// TwinCAT 3 PLC project PLC1
// ProgramVersion: 3.1.4024.0
// libraries:
//   CmpBitmapPool, * (System)
//   Tc2_Standard, * (Beckhoff Automation GmbH)
//   Tc2_System, * (Beckhoff Automation GmbH)
//   Tc3_Module, * (Beckhoff Automation GmbH)
// project tree:
//   GVLs/ GVL_UNIT_Blikkenvullijn.TcGVL
//   LIB/1. Control Modules/Brisq/1. DEV_Base/ FB_DeviceBase.TcPOU, stDevBase.TcDUT
//   LIB/1. Control Modules/Brisq/2. DEV_AnaIn/ FB_DEV_AnaIn.TcPOU, ITF_DEV_AnaIn.TcIO
//   LIB/1. Control Modules/Brisq/3. DEV_DigIn/ FB_DEV_DigIn.TcPOU, ITF_DigIn.TcIO
//   LIB/1. Control Modules/Brisq/4. DEV_Valve/ DEV_Valve.TcPOU, ITF_Valve.TcIO
//   LIB/1. Control Modules/Brisq/4. DEV_Valve/ENUMs/ E_ValveState.TcDUT
//   LIB/1. Control Modules/Brisq/4. DEV_Valve/STRUCTs/ stDevValve.TcDUT
//   LIB/1. Control Modules/Brisq/5. DEV_ControlValve/ DEV_CtrlValve.TcPOU, ITF_ControlValve.TcIO
//   LIB/1. Control Modules/Brisq/5. DEV_ControlValve/ENUMs/ E_CtrlValveState.TcDUT
//   LIB/1. Control Modules/Brisq/6. DEV_Motor/ENUMs/ E_MotorState.TcDUT
//   LIB/1. Control Modules/Brisq/6. DEV_Motor/ ITF_Motor_1.TcIO
//   LIB/1. Control Modules/Brisq/ENUMs/ E_OperationMode.TcDUT
//   LIB/1. Control Modules/Brisq/ FB_Devices.TcPOU
//   LIB/2. Equipment Modules/1. FB_Base/ FB_EMbase.TcPOU, stEMbase.TcDUT
//   LIB/2. Equipment Modules/2. EM_Machine_PackML/ FB_Machine_PackML.TcPOU, ITF_PackML.TcIO, STRUCT_Machine_PackML.TcDUT
//   LIB/3. Units/1. UN_Base/ FB_UN_base.TcPOU, stUNbase.TcDUT
//   / PlcTask.TcTTO
//   POUs/1. Control Modules/1. CM_Motor/ CM_Motor.TcPOU, ITF_Motor.TcIO
//   POUs/1. Control Modules/1. CM_Motor/Enums/ E_Motor_Error_State.TcDUT, E_Motor_State.TcDUT
//   POUs/1. Control Modules/1. CM_Motor/Structs/1. CS/ CM_Motor_CS.TcDUT
//   POUs/1. Control Modules/1. CM_Motor/Structs/2. HMI/ CM_Motor_HMI.TcDUT
//   POUs/1. Control Modules/1. CM_Motor/Structs/3. STS/ CM_Motor_STS.TcDUT
//   POUs/1. Control Modules/1. CM_Motor/Structs/4. ALM/ CM_Motor_ALM.TcDUT
//   POUs/1. Control Modules/1. CM_Motor/Structs/5. WRN/ CM_Motor_WRN.TcDUT
//   POUs/1. Control Modules/1. CM_Motor/Structs/6. PAR/ CM_Motor_PAR.TcDUT
//   POUs/1. Control Modules/1. CM_Motor/Structs/7. SIM/ CM_Motor_SIM.TcDUT
//   POUs/1. Control Modules/1. CM_Motor/Structs/ STRUCT_CM_Motor.TcDUT
//   POUs/1. Control Modules/2. CM_Sensor/ CM_Sensor.TcPOU, ITF_Sensor.TcIO
//   POUs/1. Control Modules/2. CM_Sensor/Structs/1. CS/ CM_Sensor_CS.TcDUT
//   POUs/1. Control Modules/2. CM_Sensor/Structs/2. HMI/ CM_Sensor_HMI.TcDUT
//   POUs/1. Control Modules/2. CM_Sensor/Structs/3. STS/ CM_Sensor_STS.TcDUT
//   POUs/1. Control Modules/2. CM_Sensor/Structs/4. ALM/ CM_Sensor_ALM.TcDUT
//   POUs/1. Control Modules/2. CM_Sensor/Structs/5. WRN/ CM_Sensor_WRN.TcDUT
//   POUs/1. Control Modules/2. CM_Sensor/Structs/6. PAR/ CM_Sensor_PAR.TcDUT
//   POUs/1. Control Modules/2. CM_Sensor/Structs/7. SIM/ CM_Sensor_SIM.TcDUT
//   POUs/1. Control Modules/2. CM_Sensor/Structs/ STRUCT_CM_Sensor.TcDUT
//   POUs/1. Control Modules/4. CM_Valve/ CM_Valve.TcPOU, ITF_Valve2.TcIO
//   POUs/1. Control Modules/4. CM_Valve/Enums/ E_Valve_Error_State.TcDUT, E_Valve_State.TcDUT
//   POUs/1. Control Modules/4. CM_Valve/Structs/1. CS/ CM_Valve_CS.TcDUT
//   POUs/1. Control Modules/4. CM_Valve/Structs/2. HMI/ CM_Valve_HMI.TcDUT
//   POUs/1. Control Modules/4. CM_Valve/Structs/3. STS/ CM_Valve_STS.TcDUT
//   POUs/1. Control Modules/4. CM_Valve/Structs/4. ALM/ CM_Valve_ALM.TcDUT
//   POUs/1. Control Modules/4. CM_Valve/Structs/5. WRN/ CM_Valve_WRN.TcDUT
//   POUs/1. Control Modules/4. CM_Valve/Structs/6. PAR/ CM_Valve_PAR.TcDUT
//   POUs/1. Control Modules/4. CM_Valve/Structs/7. SIM/ CM_Valve_SIM.TcDUT
//   POUs/1. Control Modules/4. CM_Valve/Structs/ STRUCT_CM_Valve.TcDUT
//   POUs/2. Equipment Modules/1. EM_Can_Supply/Enums/ E_State_Can_Supply.TcDUT
//   POUs/2. Equipment Modules/1. EM_Can_Supply/ EM_Can_Supply.TcPOU, ITF_Can_Supply.TcIO
//   POUs/2. Equipment Modules/1. EM_Can_Supply/Structs/1. CS/ EM_CanSupply_CS.TcDUT
//   POUs/2. Equipment Modules/1. EM_Can_Supply/Structs/2. HMI/ EM_CanSupply_HMI.TcDUT
//   POUs/2. Equipment Modules/1. EM_Can_Supply/Structs/3. STS/ EM_CanSupply_STS.TcDUT
//   POUs/2. Equipment Modules/1. EM_Can_Supply/Structs/4. ALM/ EM_CanSupply_ALM.TcDUT
//   POUs/2. Equipment Modules/1. EM_Can_Supply/Structs/5. WRN/ EM_CanSupply_WRN.TcDUT
//   POUs/2. Equipment Modules/1. EM_Can_Supply/Structs/6. PAR/ EM_CanSupply_PAR.TcDUT
//   POUs/2. Equipment Modules/1. EM_Can_Supply/Structs/7. SIM/ EM_CanSupply_SIM.TcDUT
//   POUs/2. Equipment Modules/1. EM_Can_Supply/Structs/ STRUCT_EM_CanSupply.TcDUT
//   POUs/2. Equipment Modules/2. EM_Filling/ EM_Filling.TcPOU
//   POUs/2. Equipment Modules/2. EM_Filling/Enums/ E_State_Filling.TcDUT
//   POUs/2. Equipment Modules/2. EM_Filling/Structs/1. CS/ EM_Filling_CS.TcDUT
//   POUs/2. Equipment Modules/2. EM_Filling/Structs/2. HMI/ EM_Filling_HMI.TcDUT
//   POUs/2. Equipment Modules/2. EM_Filling/Structs/3. STS/ EM_Filling_STS.TcDUT
//   POUs/2. Equipment Modules/2. EM_Filling/Structs/4. ALM/ EM_Filling_ALM.TcDUT
//   POUs/2. Equipment Modules/2. EM_Filling/Structs/5. WRN/ EM_Filling_WRN.TcDUT
//   POUs/2. Equipment Modules/2. EM_Filling/Structs/6. PAR/ EM_Filling_PAR.TcDUT
//   POUs/2. Equipment Modules/2. EM_Filling/Structs/7. SIM/ EM_Filling_SIM.TcDUT
//   POUs/2. Equipment Modules/2. EM_Filling/Structs/ STRUCT_EM_Filling.TcDUT
//   POUs/2. Equipment Modules/4. EM_Transport/ EM_Transport.TcPOU, ITF_EM_Transport.TcIO
//   POUs/2. Equipment Modules/4. EM_Transport/Structs/1. CS/ EM_Transport_CS.TcDUT
//   POUs/2. Equipment Modules/4. EM_Transport/Structs/2. HMI/ EM_Transport_HMI.TcDUT
//   POUs/2. Equipment Modules/4. EM_Transport/Structs/3. STS/ EM_Transport_STS.TcDUT
//   POUs/2. Equipment Modules/4. EM_Transport/Structs/4. ALM/ EM_Transport_ALM.TcDUT
//   POUs/2. Equipment Modules/4. EM_Transport/Structs/5. WRN/ EM_Transport_WRN.TcDUT
//   POUs/2. Equipment Modules/4. EM_Transport/Structs/6. PAR/ EM_Transport_PAR.TcDUT
//   POUs/2. Equipment Modules/4. EM_Transport/Structs/7. SIM/ EM_Transport_SIM.TcDUT
//   POUs/2. Equipment Modules/4. EM_Transport/Structs/ STRUCT_EM_Transport.TcDUT
//   POUs/2. Equipment Modules/3. EM_Machine/ EM_Machine.TcPOU
//   POUs/2. Equipment Modules/3. EM_Machine/Structs/1. CS/ EM_Machine_CS.TcDUT
//   POUs/2. Equipment Modules/3. EM_Machine/Structs/2. HMI/ EM_Machine_HMI.TcDUT
//   POUs/2. Equipment Modules/3. EM_Machine/Structs/3. STS/ EM_Machine_STS.TcDUT
//   POUs/2. Equipment Modules/3. EM_Machine/Structs/4. ALM/ EM_Machine_ALM.TcDUT
//   POUs/2. Equipment Modules/3. EM_Machine/Structs/5. WRN/ EM_Machine_WRN.TcDUT
//   POUs/2. Equipment Modules/3. EM_Machine/Structs/6. PAR/ EM_Machine_PAR.TcDUT
//   POUs/2. Equipment Modules/3. EM_Machine/Structs/7. SIM/ EM_Machine_SIM.TcDUT
//   POUs/2. Equipment Modules/3. EM_Machine/Structs/ STRUCT_EM_Machine.TcDUT
//   POUs/2. Equipment Modules/5. EM_Transport_Mechanische_Stop/ EM_Transport_Mechanische_Stop.TcPOU, ITF_EM_Transport_Mechanische_Stop.TcIO
//   POUs/2. Equipment Modules/5. EM_Transport_Mechanische_Stop/Enums/ E_Mechanische_Stop.TcDUT
//   POUs/2. Equipment Modules/5. EM_Transport_Mechanische_Stop/Structs/1. CS/ EM_Transport_Mechanische_Stop_CS.TcDUT
//   POUs/2. Equipment Modules/5. EM_Transport_Mechanische_Stop/Structs/2. HMI/ EM_Transport_Mechanische_Stop_HMI.TcDUT
//   POUs/2. Equipment Modules/5. EM_Transport_Mechanische_Stop/Structs/3. STS/ EM_Transport_Mechanische_Stop_STS.TcDUT
//   POUs/2. Equipment Modules/5. EM_Transport_Mechanische_Stop/Structs/4. ALM/ EM_Transport_Mechanische_Stop_ALM.TcDUT
//   POUs/2. Equipment Modules/5. EM_Transport_Mechanische_Stop/Structs/5. WRN/ EM_Transport_Mechanische_Stop_WRN.TcDUT
//   POUs/2. Equipment Modules/5. EM_Transport_Mechanische_Stop/Structs/6. PAR/ EM_Transport_Mechanische_Stop_PAR.TcDUT
//   POUs/2. Equipment Modules/5. EM_Transport_Mechanische_Stop/Structs/7. SIM/ EM_Transport_Mechanische_Stop_SIM.TcDUT
//   POUs/2. Equipment Modules/5. EM_Transport_Mechanische_Stop/Structs/ STRUCT_EM_Mechanische_Stop.TcDUT
//   POUs/3. Units/1. Unit_Blikkenvullijn/ ITF_UNIT_Blikkenvullijn.TcIO, UNIT_Blikkenvullijn.TcPOU
//   POUs/3. Units/1. Unit_Blikkenvullijn/Structs/4. ALM/ UNIT_Blikkenvullijn_ALM.TcDUT
//   POUs/3. Units/1. Unit_Blikkenvullijn/Structs/1. CS/ UNIT_Blikkenvullijn_CS.TcDUT
//   POUs/3. Units/1. Unit_Blikkenvullijn/Structs/2. HMI/ UNIT_Blikkenvullijn_HMI.TcDUT
//   POUs/3. Units/1. Unit_Blikkenvullijn/Structs/6. PAR/ UNIT_Blikkenvullijn_PAR.TcDUT
//   POUs/3. Units/1. Unit_Blikkenvullijn/Structs/7. SIM/ UNIT_Blikkenvullijn_SIM.TcDUT
//   POUs/3. Units/1. Unit_Blikkenvullijn/Structs/ STRUCT_UNIT_Blikkenvullijn.TcDUT
//   POUs/3. Units/1. Unit_Blikkenvullijn/Structs/3. STS/ UNIT_Blikkenvullijn_STS.TcDUT
//   POUs/3. Units/1. Unit_Blikkenvullijn/Structs/5. WRN/ UNIT_Blikkenvullijn_WRN.TcDUT
//   POUs/4. Management/1. AlarmHandler/ AlarmHandler.TcPOU, stErrorHandling.TcDUT
//   POUs/4. Management/2. ModeSelect/ ITF_ModeSelect.TcIO, ModeSelect.TcPOU, STRUCT_ModeSelect.TcDUT
//   POUs/4. Management/3. PackML/ E_State_PackML.TcDUT, ITF_PackMLV2.TcIO, PackML_StateMachine.TcPOU
//   POUs/ MAIN.TcPOU
// real-time tasks:
//   TASK PlcTask: cycle T#10ms, priority 20, ADS port 350

CONFIGURATION PLC1
    RESOURCE PLC ON TwinCAT3
        TASK PlcTask(INTERVAL := T#1ms, PRIORITY := 11);
        PROGRAM MAIN WITH PlcTask : MAIN;
    END_RESOURCE
END_CONFIGURATION

// ---- LIB/1. Control Modules/Brisq/1. DEV_Base/stDevBase.TcDUT
TYPE stDevBase :
STRUCT
	sTagName : STRING;
	sDescription : STRING;
END_STRUCT
END_TYPE

// ---- LIB/1. Control Modules/Brisq/4. DEV_Valve/ENUMs/E_ValveState.TcDUT
{attribute 'qualified_only'}
{attribute 'strict'}
TYPE E_ValveState :
(
	Unknown := 0,
	Open := 1,
	Closed := 2,
	Opening := 3,
	Closing := 4,
	Error := -1
);
END_TYPE

// ---- LIB/1. Control Modules/Brisq/4. DEV_Valve/STRUCTs/stDevValve.TcDUT
TYPE stDevValve :
STRUCT
	//Input to HMI
	bGetHmiError : BOOL;  //True = error
	bGetHmiStatus : BOOL; //True = Open || False = Closed
	eGetState : E_ValveState;
	eGetMode : E_OperationMode;
	
	//Output from HMI
	eSetMode : E_OperationMode; 
END_STRUCT
END_TYPE

// ---- LIB/1. Control Modules/Brisq/5. DEV_ControlValve/ENUMs/E_CtrlValveState.TcDUT
{attribute 'qualified_only'}
{attribute 'strict'}
TYPE E_CtrlValveState :
(
	Unknown := 0,
	InPosition := 1,
	Moving := 2,
	Error := -1
);
END_TYPE

// ---- LIB/1. Control Modules/Brisq/6. DEV_Motor/ENUMs/E_MotorState.TcDUT
{attribute 'qualified_only'}
{attribute 'strict'}
TYPE E_MotorState :
(
	Unknown := 0,
	Running := 1,
	Stalled := 2,
	SpeedingUp := 3,
	SpeedingDown := 4,
	Error := -1
);
END_TYPE

// ---- LIB/1. Control Modules/Brisq/ENUMs/E_OperationMode.TcDUT
{attribute 'qualified_only'}
{attribute 'strict'}
TYPE E_OperationMode :
(
	Off := 0,
	Manual := 1,
	Automatic := 2
);
END_TYPE

// ---- LIB/2. Equipment Modules/1. FB_Base/stEMbase.TcDUT
TYPE stEMbase :
STRUCT
	sTagName : STRING;
	sDescription : STRING;
END_STRUCT
END_TYPE

// ---- LIB/2. Equipment Modules/2. EM_Machine_PackML/STRUCT_Machine_PackML.TcDUT
TYPE STRUCT_Machine_PackML :
STRUCT
	//Properties
	State 			: E_State_PackML;
	//Methods
   	Abort 			: BOOL;
	Aborting_SC 	: BOOL;
	Clear 			: BOOL;
	Clearing_SC 	: BOOL;
	Execute_SC 		: BOOL;
	Completing_SC	: BOOL;
	Hold 			: BOOL;
	Holding_SC 		: BOOL;
	Reset 			: BOOL;
	Resetting_SC 	: BOOL;
	Start 			: BOOL;
	Starting_SC 	: BOOL;
	Stop 			: BOOL;
	Stopping_SC 	: BOOL;
	Suspend 		: BOOL;
	Suspending_SC 	: BOOL;
	Unhold 			: BOOL;
	Unholding_SC 	: BOOL;
	Unsuspend 		: BOOL;
	Unsuspending_SC : BOOL;
END_STRUCT
END_TYPE

// ---- LIB/3. Units/1. UN_Base/stUNbase.TcDUT
TYPE stUNbase :
STRUCT
	sTagName : STRING;
	sDescription : STRING;
END_STRUCT
END_TYPE

// ---- POUs/1. Control Modules/1. CM_Motor/Enums/E_Motor_Error_State.TcDUT
{attribute 'qualified_only'}
{attribute 'strict'}
TYPE E_Motor_Error_State :
(
	enum_member := 0
);
END_TYPE

// ---- POUs/1. Control Modules/1. CM_Motor/Enums/E_Motor_State.TcDUT
{attribute 'qualified_only'}
{attribute 'strict'}
TYPE E_Motor_State :
(
	enum_member := 0
);
END_TYPE

// ---- POUs/1. Control Modules/1. CM_Motor/Structs/1. CS/CM_Motor_CS.TcDUT
TYPE CM_Motor_CS :
STRUCT
	Start		: BOOL;
	Stop		: BOOL;
	Reset		: BOOL;
	Abort		: BOOL;
	Clear		: BOOL;
	UnSuspend	: BOOL;
	Suspend		: BOOL;
	UnHold		: BOOL;
	Hold		: BOOL;
	Richting_L	: BOOL;
	Richting_R	: BOOL;
	Toerental	: INT;
	Auto		: BOOL;
	Manueel		: BOOL;
END_STRUCT
END_TYPE

// ---- POUs/1. Control Modules/1. CM_Motor/Structs/2. HMI/CM_Motor_HMI.TcDUT
TYPE CM_Motor_HMI :
STRUCT
	Start		: BOOL;
	Stop		: BOOL;
	Reset		: BOOL;
	Abort		: BOOL;
	Clear		: BOOL;
	UnSuspend	: BOOL;
	Suspend		: BOOL;
	UnHold		: BOOL;
	Hold		: BOOL;
	Richting_L	: BOOL;
	Richting_R	: BOOL;
	Toerental	: INT;
	Auto		: BOOL;
	Manueel		: BOOL;
END_STRUCT
END_TYPE

// ---- POUs/1. Control Modules/1. CM_Motor/Structs/3. STS/CM_Motor_STS.TcDUT
TYPE CM_Motor_STS :
STRUCT
	Tag				: STRING;
	State 			: E_State_PackML;
	Error_State 	: E_Motor_Error_State;
	Richting_L		: BOOL;
	Richting_R		: BOOL;
	Auto			: BOOL;
	Manueel			: BOOL;
	Toerental 		: INT;
	
	Starting_SC		: BOOL;
	Execute_SC		: BOOL;
	Resetting_SC	: BOOL;
	Holding_SC		: BOOL;
	Unholding_SC	: BOOL;
	Suspending_SC	: BOOL;
	Unsuspending_SC	: BOOL;
	Aborting_SC		: BOOL;
	Clearing_SC		: BOOL;
	Stopping_SC		: BOOL;
	Completing_SC	: BOOL;
END_STRUCT
END_TYPE

// ---- POUs/1. Control Modules/1. CM_Motor/Structs/4. ALM/CM_Motor_ALM.TcDUT
TYPE CM_Motor_ALM :
STRUCT
END_STRUCT
END_TYPE

// ---- POUs/1. Control Modules/1. CM_Motor/Structs/5. WRN/CM_Motor_WRN.TcDUT
TYPE CM_Motor_WRN :
STRUCT
END_STRUCT
END_TYPE

// ---- POUs/1. Control Modules/1. CM_Motor/Structs/6. PAR/CM_Motor_PAR.TcDUT
TYPE CM_Motor_PAR :
STRUCT
END_STRUCT
END_TYPE

// ---- POUs/1. Control Modules/1. CM_Motor/Structs/7. SIM/CM_Motor_SIM.TcDUT
TYPE CM_Motor_SIM :
STRUCT
END_STRUCT
END_TYPE

// ---- POUs/1. Control Modules/1. CM_Motor/Structs/STRUCT_CM_Motor.TcDUT
TYPE STRUCT_CM_Motor :
STRUCT
	CS	: CM_Motor_CS;
	HMI	: CM_Motor_HMI;
	STS	: CM_Motor_STS;
	ALM	: CM_Motor_ALM;
	WRN	: CM_Motor_WRN;
	PAR	: CM_Motor_PAR;
	SIM	: CM_Motor_SIM;
END_STRUCT
END_TYPE

// ---- POUs/1. Control Modules/2. CM_Sensor/Structs/1. CS/CM_Sensor_CS.TcDUT
TYPE CM_Sensor_CS :
STRUCT
	Auto		: BOOL;
	Manueel		: BOOL;
	Output		: BOOL;
END_STRUCT
END_TYPE

// ---- POUs/1. Control Modules/2. CM_Sensor/Structs/2. HMI/CM_Sensor_HMI.TcDUT
TYPE CM_Sensor_HMI :
STRUCT
	Auto		: BOOL;
	Manueel		: BOOL;
	Output		: BOOL;
END_STRUCT
END_TYPE

// ---- POUs/1. Control Modules/2. CM_Sensor/Structs/3. STS/CM_Sensor_STS.TcDUT
TYPE CM_Sensor_STS :
STRUCT
	Tag				: STRING;
	Output			: BOOL;
	Auto			: BOOL;
	Manueel			: BOOL;
END_STRUCT
END_TYPE

// ---- POUs/1. Control Modules/2. CM_Sensor/Structs/4. ALM/CM_Sensor_ALM.TcDUT
TYPE CM_Sensor_ALM :
STRUCT
END_STRUCT
END_TYPE

// ---- POUs/1. Control Modules/2. CM_Sensor/Structs/5. WRN/CM_Sensor_WRN.TcDUT
TYPE CM_Sensor_WRN :
STRUCT
END_STRUCT
END_TYPE

// ---- POUs/1. Control Modules/2. CM_Sensor/Structs/6. PAR/CM_Sensor_PAR.TcDUT
TYPE CM_Sensor_PAR :
STRUCT
END_STRUCT
END_TYPE

// ---- POUs/1. Control Modules/2. CM_Sensor/Structs/7. SIM/CM_Sensor_SIM.TcDUT
TYPE CM_Sensor_SIM :
STRUCT
END_STRUCT
END_TYPE

// ---- POUs/1. Control Modules/2. CM_Sensor/Structs/STRUCT_CM_Sensor.TcDUT
TYPE STRUCT_CM_Sensor :
STRUCT
	CS	: CM_Sensor_CS;
	HMI	: CM_Sensor_HMI;
	STS	: CM_Sensor_STS;
	ALM	: CM_Sensor_ALM;
	WRN	: CM_Sensor_WRN;
	PAR	: CM_Sensor_PAR;
	SIM	: CM_Sensor_SIM;
END_STRUCT
END_TYPE

// ---- POUs/1. Control Modules/4. CM_Valve/Enums/E_Valve_Error_State.TcDUT
{attribute 'qualified_only'}
{attribute 'strict'}
TYPE E_Valve_Error_State :
(
	enum_member := 0
);
END_TYPE

// ---- POUs/1. Control Modules/4. CM_Valve/Enums/E_Valve_State.TcDUT
{attribute 'qualified_only'}
{attribute 'strict'}
TYPE E_Valve_State :
(
	enum_member := 0
);
END_TYPE

// ---- POUs/1. Control Modules/4. CM_Valve/Structs/1. CS/CM_Valve_CS.TcDUT
TYPE CM_Valve_CS :
STRUCT
	Start		: BOOL;
	Stop		: BOOL;
	Reset		: BOOL;
	Abort		: BOOL;
	Clear		: BOOL;
	UnSuspend	: BOOL;
	Suspend		: BOOL;
	UnHold		: BOOL;
	Hold		: BOOL;
	Auto		: BOOL;
	Manueel		: BOOL;
	Open		: BOOL;
	Close		: BOOL;
END_STRUCT
END_TYPE

// ---- POUs/1. Control Modules/4. CM_Valve/Structs/2. HMI/CM_Valve_HMI.TcDUT
TYPE CM_Valve_HMI :
STRUCT
	Start		: BOOL;
	Stop		: BOOL;
	Reset		: BOOL;
	Abort		: BOOL;
	Clear		: BOOL;
	UnSuspend	: BOOL;
	Suspend		: BOOL;
	UnHold		: BOOL;
	Hold		: BOOL;
	Auto		: BOOL;
	Manueel		: BOOL;
	Open		: BOOL;
	Close		: BOOL;
END_STRUCT
END_TYPE

// ---- POUs/1. Control Modules/4. CM_Valve/Structs/3. STS/CM_Valve_STS.TcDUT
TYPE CM_Valve_STS :
STRUCT
	Tag				: STRING;
	State 			: E_State_PackML;
	Error_State 	: E_Motor_Error_State;
	Auto			: BOOL;
	Manueel			: BOOL;
	Open			: BOOL;
	Close			: BOOL;
	
	Starting_SC		: BOOL;
	Execute_SC		: BOOL;
	Resetting_SC	: BOOL;
	Holding_SC		: BOOL;
	Unholding_SC	: BOOL;
	Suspending_SC	: BOOL;
	Unsuspending_SC	: BOOL;
	Aborting_SC		: BOOL;
	Clearing_SC		: BOOL;
	Stopping_SC		: BOOL;
	Completing_SC	: BOOL;
END_STRUCT
END_TYPE

// ---- POUs/1. Control Modules/4. CM_Valve/Structs/4. ALM/CM_Valve_ALM.TcDUT
TYPE CM_Valve_ALM :
STRUCT
END_STRUCT
END_TYPE

// ---- POUs/1. Control Modules/4. CM_Valve/Structs/5. WRN/CM_Valve_WRN.TcDUT
TYPE CM_Valve_WRN :
STRUCT
END_STRUCT
END_TYPE

// ---- POUs/1. Control Modules/4. CM_Valve/Structs/6. PAR/CM_Valve_PAR.TcDUT
TYPE CM_Valve_PAR :
STRUCT
END_STRUCT
END_TYPE

// ---- POUs/1. Control Modules/4. CM_Valve/Structs/7. SIM/CM_Valve_SIM.TcDUT
TYPE CM_Valve_SIM :
STRUCT
END_STRUCT
END_TYPE

// ---- POUs/1. Control Modules/4. CM_Valve/Structs/STRUCT_CM_Valve.TcDUT
TYPE STRUCT_CM_Valve :
STRUCT
	CS	: CM_Valve_CS;
	HMI	: CM_Valve_HMI;
	STS	: CM_Valve_STS;
	ALM	: CM_Valve_ALM;
	WRN	: CM_Valve_WRN;
	PAR	: CM_Valve_PAR;
	SIM	: CM_Valve_SIM;
END_STRUCT
END_TYPE

// ---- POUs/2. Equipment Modules/1. EM_Can_Supply/Enums/E_State_Can_Supply.TcDUT
{attribute 'qualified_only'}
{attribute 'strict'}
TYPE E_State_Can_Supply :
(
	State := 0
);
END_TYPE

// ---- POUs/2. Equipment Modules/1. EM_Can_Supply/Structs/1. CS/EM_CanSupply_CS.TcDUT
TYPE EM_CanSupply_CS :
STRUCT
	Start		: BOOL;
	Stop		: BOOL;
	Reset		: BOOL;
	Abort		: BOOL;
	Richting_L	: BOOL;
	Richting_R	: BOOL;
	Toerental	: INT;
	Auto		: BOOL;
	Manueel		: BOOL;
	Clear		: BOOL;
	UnSuspend	: BOOL;
	Suspend		: BOOL;
	UnHold		: BOOL;
	Hold		: BOOL;
END_STRUCT
END_TYPE

// ---- POUs/2. Equipment Modules/1. EM_Can_Supply/Structs/2. HMI/EM_CanSupply_HMI.TcDUT
TYPE EM_CanSupply_HMI :
STRUCT
	Start		: BOOL;
	Stop		: BOOL;
	Reset		: BOOL;
	Abort		: BOOL;
	Richting_L	: BOOL;
	Richting_R	: BOOL;
	Toerental	: INT;
	Auto		: BOOL;
	Manueel		: BOOL;
END_STRUCT
END_TYPE

// ---- POUs/2. Equipment Modules/1. EM_Can_Supply/Structs/3. STS/EM_CanSupply_STS.TcDUT
TYPE EM_CanSupply_STS :
STRUCT
	Tag				: STRING;
	State 			: E_State_PackML;
	StringState		: STRING;
	Error_State 	: E_Motor_Error_State;
	Auto			: BOOL;
	Manueel			: BOOL;
	Richting_L		: BOOL;
	Richting_R		: BOOL;
	Starting_SC 	: BOOL;
	Execute_SC 		: BOOL;
	Resetting_SC 	: BOOL;
	Holding_SC 		: BOOL;
	Unholding_SC 	: BOOL;
	Suspending_SC	: BOOL;
	Unsuspending_SC	: BOOL;
	Aborting_SC		: BOOL;
	Clearing_SC		: BOOL;
	Stopping_SC		: BOOL;
	Completing_SC	: BOOL;
END_STRUCT
END_TYPE

// ---- POUs/2. Equipment Modules/1. EM_Can_Supply/Structs/4. ALM/EM_CanSupply_ALM.TcDUT
TYPE EM_CanSupply_ALM :
STRUCT
END_STRUCT
END_TYPE

// ---- POUs/2. Equipment Modules/1. EM_Can_Supply/Structs/5. WRN/EM_CanSupply_WRN.TcDUT
TYPE EM_CanSupply_WRN :
STRUCT
END_STRUCT
END_TYPE

// ---- POUs/2. Equipment Modules/1. EM_Can_Supply/Structs/6. PAR/EM_CanSupply_PAR.TcDUT
TYPE EM_CanSupply_PAR :
STRUCT
END_STRUCT
END_TYPE

// ---- POUs/2. Equipment Modules/1. EM_Can_Supply/Structs/7. SIM/EM_CanSupply_SIM.TcDUT
TYPE EM_CanSupply_SIM :
STRUCT
	Sen_A1_Near_TRUE	: BOOL;
	Sen_A1_Far_TRUE		: BOOL;
	Sen_A2_Near_TRUE	: BOOL;
	Sen_A2_Far_TRUE		: BOOL;
END_STRUCT
END_TYPE

// ---- POUs/2. Equipment Modules/1. EM_Can_Supply/Structs/STRUCT_EM_CanSupply.TcDUT
TYPE STRUCT_EM_CanSupply :
STRUCT
	CS	: EM_CanSupply_CS;
	HMI	: EM_CanSupply_HMI;
	STS	: EM_CanSupply_STS;
	ALM	: EM_CanSupply_ALM;
	WRN	: EM_CanSupply_WRN;
	PAR	: EM_CanSupply_PAR;
	SIM	: EM_CanSupply_SIM;	
END_STRUCT
END_TYPE

// ---- POUs/2. Equipment Modules/2. EM_Filling/Enums/E_State_Filling.TcDUT
{attribute 'qualified_only'}
{attribute 'strict'}
TYPE E_State_Filling :
(
	State := 0
);
END_TYPE

// ---- POUs/2. Equipment Modules/2. EM_Filling/Structs/1. CS/EM_Filling_CS.TcDUT
TYPE EM_Filling_CS :
STRUCT
	Start		: BOOL;
	Stop		: BOOL;
	Reset		: BOOL;
	Abort		: BOOL;
	Richting_L	: BOOL;
	Richting_R	: BOOL;
	Toerental	: INT;
	Auto		: BOOL;
	Manueel		: BOOL;
	Clear		: BOOL;
	UnSuspend	: BOOL;
	Suspend		: BOOL;
	UnHold		: BOOL;
	Hold		: BOOL;
END_STRUCT
END_TYPE

// ---- POUs/2. Equipment Modules/2. EM_Filling/Structs/2. HMI/EM_Filling_HMI.TcDUT
TYPE EM_Filling_HMI :
STRUCT
	Start		: BOOL;
	Stop		: BOOL;
	Reset		: BOOL;
	Abort		: BOOL;
	Richting_L	: BOOL;
	Richting_R	: BOOL;
	Toerental	: INT;
	Auto		: BOOL;
	Manueel		: BOOL;
	Clear		: BOOL;
	UnSuspend	: BOOL;
	Suspend		: BOOL;
	UnHold		: BOOL;
	Hold		: BOOL;
END_STRUCT
END_TYPE

// ---- POUs/2. Equipment Modules/2. EM_Filling/Structs/3. STS/EM_Filling_STS.TcDUT
TYPE EM_Filling_STS :
STRUCT
	Tag				: STRING;
	State 			: E_State_PackML;
	StringState		: STRING;
	Error_State 	: E_Motor_Error_State;
	Richting_L		: BOOL;
	Richting_R		: BOOL;
	Auto 			: BOOL;
	Manueel 		: BOOL;
	Starting_SC 	: BOOL;
	Execute_SC 		: BOOL;
	Resetting_SC 	: BOOL;
	Holding_SC 		: BOOL;
	Unholding_SC 	: BOOL;
	Suspending_SC	: BOOL;
	Unsuspending_SC	: BOOL;
	Aborting_SC		: BOOL;
	Clearing_SC		: BOOL;
	Stopping_SC		: BOOL;
	Completing_SC	: BOOL;
END_STRUCT
END_TYPE

// ---- POUs/2. Equipment Modules/2. EM_Filling/Structs/4. ALM/EM_Filling_ALM.TcDUT
TYPE EM_Filling_ALM :
STRUCT
END_STRUCT
END_TYPE

// ---- POUs/2. Equipment Modules/2. EM_Filling/Structs/5. WRN/EM_Filling_WRN.TcDUT
TYPE EM_Filling_WRN :
STRUCT
END_STRUCT
END_TYPE

// ---- POUs/2. Equipment Modules/2. EM_Filling/Structs/6. PAR/EM_Filling_PAR.TcDUT
TYPE EM_Filling_PAR :
STRUCT
END_STRUCT
END_TYPE

// ---- POUs/2. Equipment Modules/2. EM_Filling/Structs/7. SIM/EM_Filling_SIM.TcDUT
TYPE EM_Filling_SIM :
STRUCT
END_STRUCT
END_TYPE

// ---- POUs/2. Equipment Modules/2. EM_Filling/Structs/STRUCT_EM_Filling.TcDUT
TYPE STRUCT_EM_Filling :
STRUCT
	CS	: EM_Filling_CS;
	HMI	: EM_Filling_HMI;
	STS	: EM_Filling_STS;
	ALM	: EM_Filling_ALM;
	WRN	: EM_Filling_WRN;
	PAR	: EM_Filling_PAR;
	SIM	: EM_Filling_SIM;	
END_STRUCT
END_TYPE

// ---- POUs/2. Equipment Modules/4. EM_Transport/Structs/1. CS/EM_Transport_CS.TcDUT
TYPE EM_Transport_CS :
STRUCT
	Start		: BOOL;
	Stop		: BOOL;
	Reset		: BOOL;
	Abort		: BOOL;
	Auto		: BOOL;
	Manueel		: BOOL;
	Clear		: BOOL;
	UnSuspend	: BOOL;
	Suspend		: BOOL;
	UnHold		: BOOL;
	Hold		: BOOL;
END_STRUCT
END_TYPE

// ---- POUs/2. Equipment Modules/4. EM_Transport/Structs/2. HMI/EM_Transport_HMI.TcDUT
TYPE EM_Transport_HMI :
STRUCT
	Start		: BOOL;
	Stop		: BOOL;
	Reset		: BOOL;
	Abort		: BOOL;
	Auto		: BOOL;
	Manueel		: BOOL;
	Clear		: BOOL;
	UnSuspend	: BOOL;
	Suspend		: BOOL;
	UnHold		: BOOL;
	Hold		: BOOL;
END_STRUCT
END_TYPE

// ---- POUs/2. Equipment Modules/4. EM_Transport/Structs/3. STS/EM_Transport_STS.TcDUT
TYPE EM_Transport_STS :
STRUCT
	Tag				: STRING;
	State 			: E_State_PackML;
	StringState		: STRING;
	Auto 			: BOOL;
	Manueel 		: BOOL;
	Starting_SC 	: BOOL;
	Execute_SC 		: BOOL;
	Resetting_SC 	: BOOL;
	Holding_SC 		: BOOL;
	Unholding_SC 	: BOOL;
	Suspending_SC	: BOOL;
	Unsuspending_SC	: BOOL;
	Aborting_SC		: BOOL;
	Clearing_SC		: BOOL;
	Stopping_SC		: BOOL;
	Completing_SC	: BOOL;
END_STRUCT
END_TYPE

// ---- POUs/2. Equipment Modules/4. EM_Transport/Structs/4. ALM/EM_Transport_ALM.TcDUT
TYPE EM_Transport_ALM :
STRUCT
END_STRUCT
END_TYPE

// ---- POUs/2. Equipment Modules/4. EM_Transport/Structs/5. WRN/EM_Transport_WRN.TcDUT
TYPE EM_Transport_WRN :
STRUCT
END_STRUCT
END_TYPE

// ---- POUs/2. Equipment Modules/4. EM_Transport/Structs/6. PAR/EM_Transport_PAR.TcDUT
TYPE EM_Transport_PAR :
STRUCT
END_STRUCT
END_TYPE

// ---- POUs/2. Equipment Modules/4. EM_Transport/Structs/7. SIM/EM_Transport_SIM.TcDUT
TYPE EM_Transport_SIM :
STRUCT
	Stopping_SC	: BOOL;
END_STRUCT
END_TYPE

// ---- POUs/2. Equipment Modules/4. EM_Transport/Structs/STRUCT_EM_Transport.TcDUT
TYPE STRUCT_EM_Transport :
STRUCT
	CS	: EM_Transport_CS;
	HMI	: EM_Transport_HMI;
	STS	: EM_Transport_STS;
	ALM	: EM_Transport_ALM;
	WRN	: EM_Transport_WRN;
	PAR	: EM_Transport_PAR;
	SIM	: EM_Transport_SIM;	
END_STRUCT
END_TYPE

// ---- POUs/2. Equipment Modules/3. EM_Machine/Structs/1. CS/EM_Machine_CS.TcDUT
TYPE EM_Machine_CS :
STRUCT
	Start		: BOOL;
	Stop		: BOOL;
	Reset		: BOOL;
	Abort		: BOOL;
	Clear		: BOOL;
	UnSuspend	: BOOL;
	Suspend		: BOOL;
	UnHold		: BOOL;
	Hold		: BOOL;
	Auto		: BOOL;
	Manueel		: BOOL;
END_STRUCT
END_TYPE

// ---- POUs/2. Equipment Modules/3. EM_Machine/Structs/2. HMI/EM_Machine_HMI.TcDUT
TYPE EM_Machine_HMI :
STRUCT
	Start		: BOOL;
	Stop		: BOOL;
	Reset		: BOOL;
	Abort		: BOOL;
	Clear		: BOOL;
	UnSuspend	: BOOL;
	Suspend		: BOOL;
	UnHold		: BOOL;
	Hold		: BOOL;
	Auto		: BOOL;
	Manueel 	: BOOL;
END_STRUCT
END_TYPE

// ---- POUs/2. Equipment Modules/3. EM_Machine/Structs/3. STS/EM_Machine_STS.TcDUT
TYPE EM_Machine_STS :
STRUCT
	State 			: E_State_PackML;
	StringState		: STRING;
	Auto 			: BOOL;
	Manueel 		: BOOL;
	Starting_SC 	: BOOL;
	Execute_SC 		: BOOL;
	Resetting_SC 	: BOOL;
	Holding_SC 		: BOOL;
	Unholding_SC 	: BOOL;
	Suspending_SC	: BOOL;
	Unsuspending_SC	: BOOL;
	Aborting_SC		: BOOL;
	Clearing_SC		: BOOL;
	Stopping_SC		: BOOL;
	Completing_SC	: BOOL;
END_STRUCT
END_TYPE

// ---- POUs/2. Equipment Modules/3. EM_Machine/Structs/4. ALM/EM_Machine_ALM.TcDUT
TYPE EM_Machine_ALM :
STRUCT
END_STRUCT
END_TYPE

// ---- POUs/2. Equipment Modules/3. EM_Machine/Structs/5. WRN/EM_Machine_WRN.TcDUT
TYPE EM_Machine_WRN :
STRUCT
END_STRUCT
END_TYPE

// ---- POUs/2. Equipment Modules/3. EM_Machine/Structs/6. PAR/EM_Machine_PAR.TcDUT
TYPE EM_Machine_PAR :
STRUCT
END_STRUCT
END_TYPE

// ---- POUs/2. Equipment Modules/3. EM_Machine/Structs/7. SIM/EM_Machine_SIM.TcDUT
TYPE EM_Machine_SIM :
STRUCT
END_STRUCT
END_TYPE

// ---- POUs/2. Equipment Modules/3. EM_Machine/Structs/STRUCT_EM_Machine.TcDUT
TYPE STRUCT_EM_Machine :
STRUCT
	CS	: EM_Machine_CS;
	HMI	: EM_Machine_HMI;
	STS	: EM_Machine_STS;
	ALM	: EM_Machine_ALM;
	WRN	: EM_Machine_WRN;
	PAR	: EM_Machine_PAR;
	SIM	: EM_Machine_SIM;
END_STRUCT
END_TYPE

// ---- POUs/2. Equipment Modules/5. EM_Transport_Mechanische_Stop/Enums/E_Mechanische_Stop.TcDUT
{attribute 'qualified_only'}
{attribute 'strict'}
TYPE E_Mechanische_Stop :
(
	enum_member := 0
);
END_TYPE

// ---- POUs/2. Equipment Modules/5. EM_Transport_Mechanische_Stop/Structs/1. CS/EM_Transport_Mechanische_Stop_CS.TcDUT
TYPE EM_Transport_Mechanische_Stop_CS :
STRUCT
	Start		: BOOL;
	Stop		: BOOL;
	Reset		: BOOL;
	Abort		: BOOL;
	Auto		: BOOL;
	Manueel		: BOOL;
END_STRUCT
END_TYPE

// ---- POUs/2. Equipment Modules/5. EM_Transport_Mechanische_Stop/Structs/2. HMI/EM_Transport_Mechanische_Stop_HMI.TcDUT
TYPE EM_Transport_Mechanische_Stop_HMI :
STRUCT
	Start		: BOOL;
	Stop		: BOOL;
	Reset		: BOOL;
	Abort		: BOOL;
	Auto		: BOOL;
	Manueel		: BOOL;
END_STRUCT
END_TYPE

// ---- POUs/2. Equipment Modules/5. EM_Transport_Mechanische_Stop/Structs/3. STS/EM_Transport_Mechanische_Stop_STS.TcDUT
TYPE EM_Transport_Mechanische_Stop_STS :
STRUCT
	Tag				: STRING;
	State 			: E_Mechanische_Stop;
	State2			: E_State_PackML := E_State_PackML.STOPPED;
	Manueel			: BOOL;
	Auto			: BOOL;
END_STRUCT
END_TYPE

// ---- POUs/2. Equipment Modules/5. EM_Transport_Mechanische_Stop/Structs/4. ALM/EM_Transport_Mechanische_Stop_ALM.TcDUT
TYPE EM_Transport_Mechanische_Stop_ALM :
STRUCT
END_STRUCT
END_TYPE

// ---- POUs/2. Equipment Modules/5. EM_Transport_Mechanische_Stop/Structs/5. WRN/EM_Transport_Mechanische_Stop_WRN.TcDUT
TYPE EM_Transport_Mechanische_Stop_WRN :
STRUCT
END_STRUCT
END_TYPE

// ---- POUs/2. Equipment Modules/5. EM_Transport_Mechanische_Stop/Structs/6. PAR/EM_Transport_Mechanische_Stop_PAR.TcDUT
TYPE EM_Transport_Mechanische_Stop_PAR :
STRUCT
END_STRUCT
END_TYPE

// ---- POUs/2. Equipment Modules/5. EM_Transport_Mechanische_Stop/Structs/7. SIM/EM_Transport_Mechanische_Stop_SIM.TcDUT
TYPE EM_Transport_Mechanische_Stop_SIM :
STRUCT
END_STRUCT
END_TYPE

// ---- POUs/2. Equipment Modules/5. EM_Transport_Mechanische_Stop/Structs/STRUCT_EM_Mechanische_Stop.TcDUT
TYPE STRUCT_EM_Mechanische_Stop :
STRUCT
	CS	: EM_Transport_Mechanische_Stop_CS;
	HMI	: EM_Transport_Mechanische_Stop_HMI;
	STS	: EM_Transport_Mechanische_Stop_STS;
	ALM	: EM_Transport_Mechanische_Stop_ALM;
	WRN	: EM_Transport_Mechanische_Stop_WRN;
	PAR	: EM_Transport_Mechanische_Stop_PAR;
	SIM	: EM_Transport_Mechanische_Stop_SIM;	
END_STRUCT
END_TYPE

// ---- POUs/3. Units/1. Unit_Blikkenvullijn/Structs/4. ALM/UNIT_Blikkenvullijn_ALM.TcDUT
TYPE UNIT_Blikkenvullijn_ALM :
STRUCT
END_STRUCT
END_TYPE

// ---- POUs/3. Units/1. Unit_Blikkenvullijn/Structs/1. CS/UNIT_Blikkenvullijn_CS.TcDUT
TYPE UNIT_Blikkenvullijn_CS :
STRUCT
	Start		: BOOL;
	Stop		: BOOL;
	Reset		: BOOL;
	Abort		: BOOL;
	Clear		: BOOL;
	UnSuspend	: BOOL;
	Suspend		: BOOL;
	UnHold		: BOOL;
	Hold		: BOOL;
	Auto		: BOOL;
	Manueel		: BOOL;
END_STRUCT
END_TYPE

// ---- POUs/3. Units/1. Unit_Blikkenvullijn/Structs/2. HMI/UNIT_Blikkenvullijn_HMI.TcDUT
TYPE UNIT_Blikkenvullijn_HMI :
STRUCT
	Start		: BOOL;
	Stop		: BOOL;
	Reset		: BOOL;
	Abort		: BOOL;
	Clear		: BOOL;
	UnSuspend	: BOOL;
	Suspend		: BOOL;
	UnHold		: BOOL;
	Hold		: BOOL;
	Auto		: BOOL;
	Manueel 	: BOOL;
END_STRUCT
END_TYPE

// ---- POUs/3. Units/1. Unit_Blikkenvullijn/Structs/6. PAR/UNIT_Blikkenvullijn_PAR.TcDUT
TYPE UNIT_Blikkenvullijn_PAR :
STRUCT
END_STRUCT
END_TYPE

// ---- POUs/3. Units/1. Unit_Blikkenvullijn/Structs/7. SIM/UNIT_Blikkenvullijn_SIM.TcDUT
TYPE UNIT_Blikkenvullijn_SIM :
STRUCT
	Starting_SC 	: BOOL;
	Execute_SC 		: BOOL;
	Resetting_SC 	: BOOL;
	Holding_SC 		: BOOL;
	Unholding_SC 	: BOOL;
	Suspending_SC	: BOOL;
	Unsuspending_SC	: BOOL;
	Aborting_SC		: BOOL;
	Clearing_SC		: BOOL;
	Stopping_SC		: BOOL;
END_STRUCT
END_TYPE

// ---- POUs/3. Units/1. Unit_Blikkenvullijn/Structs/STRUCT_UNIT_Blikkenvullijn.TcDUT
TYPE STRUCT_UNIT_Blikkenvullijn :
STRUCT
	CS	: UNIT_Blikkenvullijn_CS;
	HMI	: UNIT_Blikkenvullijn_HMI;
	STS	: UNIT_Blikkenvullijn_STS;
	ALM	: UNIT_Blikkenvullijn_ALM;
	WRN	: UNIT_Blikkenvullijn_WRN;
	PAR	: UNIT_Blikkenvullijn_PAR;
	SIM	: UNIT_Blikkenvullijn_SIM;
END_STRUCT
END_TYPE

// ---- POUs/3. Units/1. Unit_Blikkenvullijn/Structs/3. STS/UNIT_Blikkenvullijn_STS.TcDUT
TYPE UNIT_Blikkenvullijn_STS :
STRUCT
	State 			: E_State_PackML;
	StringState		: STRING;
	Auto 			: BOOL;
	Manueel 		: BOOL;
	Starting_SC 	: BOOL;
	Execute_SC 		: BOOL;
	Resetting_SC 	: BOOL;
	Holding_SC 		: BOOL;
	Unholding_SC 	: BOOL;
	Suspending_SC	: BOOL;
	Unsuspending_SC	: BOOL;
	Aborting_SC		: BOOL;
	Clearing_SC		: BOOL;
	Stopping_SC		: BOOL;
	Completing_SC	: BOOL;
END_STRUCT
END_TYPE

// ---- POUs/3. Units/1. Unit_Blikkenvullijn/Structs/5. WRN/UNIT_Blikkenvullijn_WRN.TcDUT
TYPE UNIT_Blikkenvullijn_WRN :
STRUCT
END_STRUCT
END_TYPE

// ---- POUs/4. Management/1. AlarmHandler/stErrorHandling.TcDUT
TYPE stErrorHandling :
STRUCT
	sTag: STRING;
	sMessage: STRING;
	sPriority: INT;
	sDevice: STRING;
	dErrorTime: DATE_AND_TIME;
	bIsAlarmAcknowledged : BOOL;
	bAcknowledged: BOOL;
	sPossibleSolution: STRING;
END_STRUCT
END_TYPE

// ---- POUs/4. Management/2. ModeSelect/STRUCT_ModeSelect.TcDUT
TYPE STRUCT_ModeSelect :
STRUCT
	Auto	: BOOL;
	Manueel	: BOOL;
	Tag		: STRING;
END_STRUCT
END_TYPE

// ---- POUs/4. Management/3. PackML/E_State_PackML.TcDUT
{attribute 'qualified_only'}
{attribute 'strict'}
{attribute 'to_string'}
TYPE E_State_PackML :
(
	STOPPED := 1,
	IDLE,
	STARTING,
	EXECUTE,
	COMPLETING,
	COMPLETE,
	RESETTING,
	HOLDING,
	HELD,
	UNHOLDING,
	SUSPENDING,
	SUSPENDED,
	UNSUSPENDING,
	ABORTING,
	ABORTED,
	CLEARING,
	STOPPING
);
END_TYPE

// ---- GVLs/GVL_UNIT_Blikkenvullijn.TcGVL
{attribute 'qualified_only'}
VAR_GLOBAL
END_VAR

// ---- LIB/1. Control Modules/Brisq/2. DEV_AnaIn/ITF_DEV_AnaIn.TcIO
INTERFACE ITF_DEV_AnaIn

END_INTERFACE

// ---- LIB/1. Control Modules/Brisq/3. DEV_DigIn/ITF_DigIn.TcIO
INTERFACE ITF_DigIn

PROPERTY ActualValue : BOOL
GET
END_GET
SET
END_SET
END_PROPERTY

PROPERTY FallingEdge : BOOL
GET
END_GET
SET
END_SET
END_PROPERTY

METHOD FB_init : BOOL
VAR_INPUT
	bInitRetains : BOOL; // if TRUE, the retain variables are initialized (warm start / cold start)
	bInCopyCode : BOOL;  // if TRUE, the instance afterwards gets moved into the copy code (online change)
END_VAR
END_METHOD

METHOD Force : BOOL
VAR_INPUT
	ForceValue : BOOL;
END_VAR
END_METHOD

METHOD ResetForce : BOOL
VAR_INPUT
END_VAR
END_METHOD

PROPERTY RisingEdge : BOOL
GET
END_GET
SET
END_SET
END_PROPERTY

END_INTERFACE

// ---- LIB/1. Control Modules/Brisq/4. DEV_Valve/ITF_Valve.TcIO
INTERFACE ITF_Valve

PROPERTY ActualState : E_ValveState
GET
END_GET
END_PROPERTY

METHOD Close : BOOL
VAR_INPUT
END_VAR
END_METHOD

PROPERTY EmergencyStatus : BOOL
GET
END_GET
END_PROPERTY

METHOD Open : BOOL
VAR_INPUT
END_VAR
END_METHOD

PROPERTY OperatingMode : BOOL
GET
END_GET
END_PROPERTY

METHOD Reset : BOOL
VAR_INPUT
END_VAR
END_METHOD

METHOD SetMode : BOOL
VAR_INPUT
END_VAR
END_METHOD

END_INTERFACE

// ---- LIB/1. Control Modules/Brisq/5. DEV_ControlValve/ITF_ControlValve.TcIO
INTERFACE ITF_ControlValve

PROPERTY EmergencyStatus : BOOL
GET
END_GET
END_PROPERTY

PROPERTY OperatingMode : BOOL
GET
END_GET
END_PROPERTY

PROPERTY OutputValue : REAL
GET
END_GET
END_PROPERTY

METHOD Reset : BOOL
VAR_INPUT
END_VAR
END_METHOD

METHOD SetMode : BOOL
VAR_INPUT
END_VAR
END_METHOD

METHOD SetValue : BOOL
VAR_INPUT
END_VAR
END_METHOD

END_INTERFACE

// ---- LIB/1. Control Modules/Brisq/6. DEV_Motor/ITF_Motor_1.TcIO
INTERFACE ITF_Motor_1

PROPERTY ActualState : BOOL
GET
END_GET
END_PROPERTY

METHOD Auto : BOOL
VAR_INPUT
END_VAR
END_METHOD

PROPERTY Error_State : BOOL
GET
END_GET
END_PROPERTY

METHOD Manueel : BOOL
VAR_INPUT
END_VAR
END_METHOD

METHOD Reset : BOOL
VAR_INPUT
END_VAR
END_METHOD

METHOD Richting_L : BOOL
VAR_INPUT
END_VAR
END_METHOD

METHOD Richting_R : BOOL
VAR_INPUT
END_VAR
END_METHOD

METHOD Start : BOOL
VAR_INPUT
END_VAR
END_METHOD

PROPERTY State : E_MotorState
GET
END_GET
END_PROPERTY

METHOD Stop : BOOL
VAR_INPUT
END_VAR
END_METHOD

METHOD Toerental : INT
VAR_INPUT
END_VAR
END_METHOD

END_INTERFACE

// ---- LIB/2. Equipment Modules/2. EM_Machine_PackML/ITF_PackML.TcIO
INTERFACE ITF_PackML

METHOD Abort : BOOL
VAR_INPUT
END_VAR
END_METHOD

METHOD Aborting_SC : BOOL
VAR_INPUT
END_VAR
END_METHOD

METHOD Clear : BOOL
VAR_INPUT
END_VAR
END_METHOD

METHOD Clearing_SC : BOOL
VAR_INPUT
END_VAR
END_METHOD

METHOD Completing_SC : BOOL
VAR_INPUT
END_VAR
END_METHOD

METHOD Execute_SC : BOOL
VAR_INPUT
END_VAR
END_METHOD

{warning 'add method implementation '}
METHOD FB_init : BOOL
VAR_INPUT
	(* if TRUE, the retain variables are initialized (warm start / cold start)*)
	bInitRetains	: BOOL;
	(* if TRUE, the instance afterwards gets moved into the copy code (online change)*)
	bInCopyCode	: BOOL;
END_VAR
END_METHOD

METHOD Hold : BOOL
VAR_INPUT
END_VAR
END_METHOD

METHOD Holding_SC : BOOL
VAR_INPUT
END_VAR
END_METHOD

METHOD Reset : BOOL
VAR_INPUT
END_VAR
END_METHOD

METHOD Resetting_SC : BOOL
VAR_INPUT
END_VAR
END_METHOD

METHOD Start : BOOL
VAR_INPUT
END_VAR
END_METHOD

METHOD Starting_SC : BOOL
VAR_INPUT
END_VAR
END_METHOD

PROPERTY State : E_State_PackML
GET
END_GET
END_PROPERTY

METHOD Stop : BOOL
VAR_INPUT
END_VAR
END_METHOD

METHOD Stopping_SC : BOOL
VAR_INPUT
END_VAR
END_METHOD

METHOD Suspend : BOOL
VAR_INPUT
END_VAR
END_METHOD

METHOD Suspending_SC : BOOL
VAR_INPUT
END_VAR
END_METHOD

METHOD Unhold : BOOL
VAR_INPUT
END_VAR
END_METHOD

METHOD Unholding_SC : BOOL
VAR_INPUT
END_VAR
END_METHOD

METHOD Unsuspend : BOOL
VAR_INPUT
END_VAR
END_METHOD

METHOD Unsuspending_SC : BOOL
VAR_INPUT
END_VAR
END_METHOD

METHOD ZeroAllVar : BOOL
VAR_INPUT
END_VAR
END_METHOD

END_INTERFACE

// ---- POUs/1. Control Modules/1. CM_Motor/ITF_Motor.TcIO
INTERFACE ITF_Motor

METHOD Abort : BOOL
VAR_INPUT
END_VAR
END_METHOD

PROPERTY Auto : BOOL
GET
END_GET
SET
END_SET
END_PROPERTY

METHOD Clear : BOOL
VAR_INPUT
END_VAR
END_METHOD

PROPERTY Error_State  : E_Motor_Error_State
GET
END_GET
END_PROPERTY

PROPERTY Manueel : BOOL
GET
END_GET
SET
END_SET
END_PROPERTY

METHOD Reset : BOOL
VAR_INPUT
END_VAR
END_METHOD

PROPERTY Richting_L : BOOL
GET
END_GET
SET
END_SET
END_PROPERTY

PROPERTY Richting_R : BOOL
GET
END_GET
SET
END_SET
END_PROPERTY

METHOD Start : BOOL
VAR_INPUT
END_VAR
END_METHOD

PROPERTY State : E_Motor_State
GET
END_GET
END_PROPERTY

METHOD Stop : BOOL
VAR_INPUT
END_VAR
END_METHOD

PROPERTY Tag : STRING
GET
END_GET
END_PROPERTY

METHOD Toerental : INT
VAR_INPUT
END_VAR
END_METHOD

END_INTERFACE

// ---- POUs/1. Control Modules/2. CM_Sensor/ITF_Sensor.TcIO
INTERFACE ITF_Sensor

PROPERTY Auto : BOOl
GET
END_GET
SET
END_SET
END_PROPERTY

PROPERTY Manueel : BOOl
GET
END_GET
SET
END_SET
END_PROPERTY

PROPERTY Output : BOOl
GET
END_GET
SET
END_SET
END_PROPERTY

PROPERTY Tag : STRING
GET
END_GET
END_PROPERTY

END_INTERFACE

// ---- POUs/1. Control Modules/4. CM_Valve/ITF_Valve2.TcIO
INTERFACE ITF_Valve2

METHOD Abort : BOOL
VAR_INPUT
END_VAR
END_METHOD

PROPERTY Auto : BOOL
GET
END_GET
SET
END_SET
END_PROPERTY

METHOD Clear : BOOL
VAR_INPUT
END_VAR
END_METHOD

METHOD Close : BOOL
VAR_INPUT
END_VAR
END_METHOD

PROPERTY Error_State  : E_Motor_Error_State
GET
END_GET
END_PROPERTY

PROPERTY Manueel : BOOL
GET
END_GET
SET
END_SET
END_PROPERTY

METHOD Open : BOOL
VAR_INPUT
END_VAR
END_METHOD

METHOD Reset : BOOL
VAR_INPUT
END_VAR
END_METHOD

METHOD Start : BOOL
VAR_INPUT
END_VAR
END_METHOD

PROPERTY State : E_Motor_State
GET
END_GET
END_PROPERTY

METHOD Stop : BOOL
VAR_INPUT
END_VAR
END_METHOD

PROPERTY Tag : STRING
GET
END_GET
END_PROPERTY

END_INTERFACE

// ---- POUs/2. Equipment Modules/1. EM_Can_Supply/ITF_Can_Supply.TcIO
INTERFACE ITF_Can_Supply EXTENDS ITF_PackML

{warning 'add method implementation '}
METHOD Abort : BOOL
END_METHOD

{warning 'add method implementation '}
METHOD Aborting_SC : BOOL
END_METHOD

{warning 'add method implementation '}
METHOD Auto : BOOL
END_METHOD

{warning 'add method implementation '}
METHOD Clear : BOOL
END_METHOD

{warning 'add method implementation '}
METHOD Clearing_SC : BOOL
END_METHOD

{warning 'add method implementation '}
METHOD Completing_SC : BOOL
END_METHOD

{warning 'add method implementation '}
METHOD Execute_SC : BOOL
END_METHOD

{warning 'add method implementation '}
METHOD FB_init : BOOL
VAR_INPUT
	bInitRetains : BOOL; // if TRUE, the retain variables are initialized (warm start / cold start)
	bInCopyCode : BOOL;  // if TRUE, the instance afterwards gets moved into the copy code (online change)
END_VAR
END_METHOD

{warning 'add method implementation '}
METHOD Hold : BOOL
END_METHOD

{warning 'add method implementation '}
METHOD Holding_SC : BOOL
END_METHOD

{warning 'add method implementation '}
METHOD Manueel : BOOL
END_METHOD

{warning 'add method implementation '}
METHOD Reset : BOOL
END_METHOD

{warning 'add method implementation '}
METHOD Resetting_SC : BOOL
END_METHOD

{warning 'add method implementation '}
METHOD Start : BOOL
END_METHOD

{warning 'add method implementation '}
METHOD Starting_SC : BOOL
END_METHOD

{warning 'add property implementation'}
PROPERTY State : E_State_PackML
GET
END_GET
END_PROPERTY

{warning 'add method implementation '}
METHOD Stop : BOOL
END_METHOD

{warning 'add method implementation '}
METHOD Stopping_SC : BOOL
END_METHOD

{warning 'add method implementation '}
METHOD Suspend : BOOL
END_METHOD

{warning 'add method implementation '}
METHOD Suspending_SC : BOOL
END_METHOD

{warning 'add method implementation '}
METHOD Unhold : BOOL
END_METHOD

{warning 'add method implementation '}
METHOD Unholding_SC : BOOL
END_METHOD

{warning 'add method implementation '}
METHOD Unsuspend : BOOL
END_METHOD

{warning 'add method implementation '}
METHOD Unsuspending_SC : BOOL
END_METHOD

{warning 'add method implementation '}
METHOD ZeroAllVar : BOOL
END_METHOD

END_INTERFACE

// ---- POUs/2. Equipment Modules/4. EM_Transport/ITF_EM_Transport.TcIO
INTERFACE ITF_EM_Transport

METHOD Abort : BOOL
VAR_INPUT
END_VAR
END_METHOD

{warning 'add method implementation '}
METHOD Auto : BOOL
END_METHOD

{warning 'add method implementation '}
METHOD Manueel : BOOL
END_METHOD

METHOD Reset : BOOL
VAR_INPUT
END_VAR
END_METHOD

PROPERTY RPM : INT
GET
END_GET
SET
END_SET
END_PROPERTY

METHOD Start : BOOL
VAR_INPUT
END_VAR
END_METHOD

PROPERTY State : E_State_PackML
GET
END_GET
END_PROPERTY

METHOD Stop : BOOL
VAR_INPUT
END_VAR
END_METHOD

PROPERTY Tag : STRING
GET
END_GET
END_PROPERTY

METHOD ZeroAllVar : BOOL
VAR_INPUT
END_VAR
END_METHOD

END_INTERFACE

// ---- POUs/2. Equipment Modules/5. EM_Transport_Mechanische_Stop/ITF_EM_Transport_Mechanische_Stop.TcIO
INTERFACE ITF_EM_Transport_Mechanische_Stop

METHOD Close : BOOL
VAR_INPUT
END_VAR
END_METHOD

METHOD Open : BOOL
VAR_INPUT
END_VAR
END_METHOD

PROPERTY Stop_State : E_Mechanische_Stop
GET
END_GET
END_PROPERTY

METHOD ZeroAllValues : BOOL
VAR_INPUT
END_VAR
END_METHOD

END_INTERFACE

// ---- POUs/3. Units/1. Unit_Blikkenvullijn/ITF_UNIT_Blikkenvullijn.TcIO
INTERFACE ITF_UNIT_Blikkenvullijn

METHOD Auto : BOOL
VAR_INPUT
END_VAR
END_METHOD

METHOD FB_init : BOOL
VAR_INPUT
	bInitRetains : BOOL; // if TRUE, the retain variables are initialized (warm start / cold start)
	bInCopyCode : BOOL;  // if TRUE, the instance afterwards gets moved into the copy code (online change)
END_VAR
END_METHOD

METHOD Manueel : BOOL
VAR_INPUT
END_VAR
END_METHOD

END_INTERFACE

// ---- POUs/4. Management/2. ModeSelect/ITF_ModeSelect.TcIO
INTERFACE ITF_ModeSelect

METHOD Auto : BOOL
VAR_INPUT
END_VAR
END_METHOD

METHOD Manueel : BOOL
VAR_INPUT
END_VAR
END_METHOD

PROPERTY Tag : STRING
GET
END_GET
SET
END_SET
END_PROPERTY

END_INTERFACE

// ---- POUs/4. Management/3. PackML/ITF_PackMLV2.TcIO
INTERFACE ITF_PackMLV2

{warning 'add method implementation '}
METHOD Abort : BOOL
END_METHOD

{warning 'add method implementation '}
METHOD Auto : BOOL
END_METHOD

{warning 'add method implementation '}
METHOD Clear : BOOL
END_METHOD

{warning 'add method implementation '}
METHOD Hold : BOOL
END_METHOD

{warning 'add method implementation '}
METHOD Manueel : BOOL
END_METHOD

{warning 'add method implementation '}
METHOD Reset : BOOL
END_METHOD

{warning 'add method implementation '}
METHOD Start : BOOL
END_METHOD

{warning 'add property implementation'}
PROPERTY State : E_State_PackML
GET
END_GET
END_PROPERTY

{warning 'add method implementation '}
METHOD Stop : BOOL
END_METHOD

{warning 'add method implementation '}
METHOD Suspend : BOOL
END_METHOD

{warning 'add method implementation '}
METHOD Unhold : BOOL
END_METHOD

{warning 'add method implementation '}
METHOD Unsuspend : BOOL
END_METHOD

{warning 'add method implementation '}
METHOD ZeroAllVar : BOOL
END_METHOD

END_INTERFACE

// ---- POUs/MAIN.TcPOU
PROGRAM MAIN
VAR
	bFirstCycleExecuted : BOOL := FALSE;
	Unit : UNIT_Blikkenvullijn;
//	Devices : FB_Devices;
	
	Start		: BOOL;
	Stop		: BOOL;
	Reset		: BOOL;
	Abort		: BOOL;
	Clear		: BOOL;
	UnSuspend	: BOOL;
	Suspend		: BOOL;
	UnHold		: BOOL;
	Hold		: BOOL;
	Auto		: BOOL;
	Manueel		: BOOL;
END_VAR

(*
$$$$$$$$\                                                                   $$\       $$$$$$$$\                     $$\                                         $$\                     
$$  _____|                                                                  $$ |      $$  _____|                    \__|                                        \__|                    
$$ |   $$$$$$\   $$$$$$\  $$$$$$$\  $$\  $$\  $$\  $$$$$$\   $$$$$$\   $$$$$$$ |      $$ |      $$$$$$$\   $$$$$$\  $$\ $$$$$$$\   $$$$$$\   $$$$$$\   $$$$$$\  $$\ $$$$$$$\   $$$$$$\  
$$$$$\ \____$$\ $$  __$$\ $$  __$$\ $$ | $$ | $$ |$$  __$$\ $$  __$$\ $$  __$$ |      $$$$$\    $$  __$$\ $$  __$$\ $$ |$$  __$$\ $$  __$$\ $$  __$$\ $$  __$$\ $$ |$$  __$$\ $$  __$$\ 
$$  __|$$$$$$$ |$$ |  \__|$$ |  $$ |$$ | $$ | $$ |$$ /  $$ |$$ /  $$ |$$ /  $$ |      $$  __|   $$ |  $$ |$$ /  $$ |$$ |$$ |  $$ |$$$$$$$$ |$$$$$$$$ |$$ |  \__|$$ |$$ |  $$ |$$ /  $$ |
$$ |  $$  __$$ |$$ |      $$ |  $$ |$$ | $$ | $$ |$$ |  $$ |$$ |  $$ |$$ |  $$ |      $$ |      $$ |  $$ |$$ |  $$ |$$ |$$ |  $$ |$$   ____|$$   ____|$$ |      $$ |$$ |  $$ |$$ |  $$ |
$$ |  \$$$$$$$ |$$ |      $$ |  $$ |\$$$$$\$$$$  |\$$$$$$  |\$$$$$$  |\$$$$$$$ |      $$$$$$$$\ $$ |  $$ |\$$$$$$$ |$$ |$$ |  $$ |\$$$$$$$\ \$$$$$$$\ $$ |      $$ |$$ |  $$ |\$$$$$$$ |
\__|   \_______|\__|      \__|  \__| \_____\____/  \______/  \______/  \_______|      \________|\__|  \__| \____$$ |\__|\__|  \__| \_______| \_______|\__|      \__|\__|  \__| \____$$ |
                                                                                                          $$\   $$ |                                                          $$\   $$ |
                                                                                                          \$$$$$$  |                                                          \$$$$$$  |
                                                                                                           \______/                                                            \______/ 
*)

//*****************************UNIT*****************************//
Unit();

//******************************CM******************************//
//Devices();


IF NOT bFirstCycleExecuted THEN
	//Unit
	Unit.FB_init(0,0);
	unit.Auto();	
	bFirstCycleExecuted := TRUE;
END_IF




    // Implement automatic mode logic
IF Start THEN
	unit.start();
	Start := FALSE;
END_IF
    
IF Stop THEN
	unit.stop();
	Stop := FALSE;
END_IF

IF Reset THEN
	Unit.reset();
	Reset := FALSE;
END_IF

IF Abort THEN
	unit.abort();
	Abort := FALSE;
END_IF

IF Clear THEN
	unit.clear();
	Clear := FALSE;
END_IF

IF UnSuspend THEN
	unit.unsuspend();
	UnSuspend := FALSE;
END_IF

IF Suspend THEN
	unit.suspend();
	Suspend := FALSE;
END_IF

IF UnHold THEN
	unit.unhold();
	UnHold := FALSE;
END_IF

IF Hold THEN
	unit.hold();
	Hold := FALSE;
END_IF

IF Auto THEN
	unit.Auto();
	Auto := FALSE;
END_IF

IF Manueel THEN
	unit.Manueel();
	Manueel := FALSE;
END_IF

END_PROGRAM

// ---- POUs/3. Units/1. Unit_Blikkenvullijn/UNIT_Blikkenvullijn.TcPOU
FUNCTION_BLOCK UNIT_Blikkenvullijn IMPLEMENTS  ITF_UNIT_Blikkenvullijn, ITF_PackMLV2
VAR
	fb_mem									: STRUCT_UNIT_Blikkenvullijn;
	bFirstCycleExecuted						: BOOL;
	
	//Custom logic
	EM_Can_Supply 							: EM_Can_Supply;	//To be programmed
	EM_Filling								: EM_Filling;		//To be tested
	CM_TurningDevice						: CM_Motor;			//To be programmed
	CM_Outfeed_ProductionLineSensor			: CM_Sensor;		//To be Tested
	
	//PackML machine's
	EM_CheckWeigher							: EM_Machine;		//Tested
	EM_BottomSeal							: EM_Machine;		//Tested
	EM_Labeller								: EM_Machine;		//Tested
	EM_TurningDevice						: EM_Machine;		//Tested
	EM_StampUnit							: EM_Machine;		//Tested
	EM_SealShrink							: EM_Machine;		//Tested
	
	//Transport logic
	EM_Infeed_CheckWeigher					: EM_Transport;			//To be tested
	EM_Transport_Checkweigher_BottomSeal	: EM_Transport;			//To be tested
	EM_Transport_BottomSeal_Labeller		: EM_Transport;			//To be tested
	EM_Transport_TurningDevice_StampUnit	: EM_Transport;			//To be tested
	EM_Transport_StampUnit_SealShrink		: EM_Transport;			//To be tested
	
	//Management Logic
	AlarmHandler 							: AlarmHandler;
	ModeSelect								: ModeSelect;
END_VAR

(*
$$$$$$$$\                                                                   $$\       $$$$$$$$\                     $$\                                         $$\                     
$$  _____|                                                                  $$ |      $$  _____|                    \__|                                        \__|                    
$$ |   $$$$$$\   $$$$$$\  $$$$$$$\  $$\  $$\  $$\  $$$$$$\   $$$$$$\   $$$$$$$ |      $$ |      $$$$$$$\   $$$$$$\  $$\ $$$$$$$\   $$$$$$\   $$$$$$\   $$$$$$\  $$\ $$$$$$$\   $$$$$$\  
$$$$$\ \____$$\ $$  __$$\ $$  __$$\ $$ | $$ | $$ |$$  __$$\ $$  __$$\ $$  __$$ |      $$$$$\    $$  __$$\ $$  __$$\ $$ |$$  __$$\ $$  __$$\ $$  __$$\ $$  __$$\ $$ |$$  __$$\ $$  __$$\ 
$$  __|$$$$$$$ |$$ |  \__|$$ |  $$ |$$ | $$ | $$ |$$ /  $$ |$$ /  $$ |$$ /  $$ |      $$  __|   $$ |  $$ |$$ /  $$ |$$ |$$ |  $$ |$$$$$$$$ |$$$$$$$$ |$$ |  \__|$$ |$$ |  $$ |$$ /  $$ |
$$ |  $$  __$$ |$$ |      $$ |  $$ |$$ | $$ | $$ |$$ |  $$ |$$ |  $$ |$$ |  $$ |      $$ |      $$ |  $$ |$$ |  $$ |$$ |$$ |  $$ |$$   ____|$$   ____|$$ |      $$ |$$ |  $$ |$$ |  $$ |
$$ |  \$$$$$$$ |$$ |      $$ |  $$ |\$$$$$\$$$$  |\$$$$$$  |\$$$$$$  |\$$$$$$$ |      $$$$$$$$\ $$ |  $$ |\$$$$$$$ |$$ |$$ |  $$ |\$$$$$$$\ \$$$$$$$\ $$ |      $$ |$$ |  $$ |\$$$$$$$ |
\__|   \_______|\__|      \__|  \__| \_____\____/  \______/  \______/  \_______|      \________|\__|  \__| \____$$ |\__|\__|  \__| \_______| \_______|\__|      \__|\__|  \__| \____$$ |
                                                                                                          $$\   $$ |                                                          $$\   $$ |
                                                                                                          \$$$$$$  |                                                          \$$$$$$  |
                                                                                                           \______/                                                            \______/ 
*)
//********************************Init PackML***********************************
fb_mem.STS.State := PackML_StateMachine(State			:= fb_mem.STS.State,
										Start           := fb_mem.CS.Start,
										Stop            := fb_mem.CS.Stop,
										Reset           := fb_mem.CS.Reset,
										Abort           := fb_mem.CS.Abort,
										Clear           := fb_mem.CS.Clear,
										UnSuspend       := fb_mem.CS.UnSuspend,
										Suspend         := fb_mem.CS.Suspend,
										UnHold          := fb_mem.CS.UnHold,
										Hold            := fb_mem.CS.Hold,
										Starting_SC     := fb_mem.STS.Starting_SC,
										Execute_SC      := fb_mem.STS.Execute_SC,
										Completing_SC	:= fb_mem.STS.Completing_SC,
										Resetting_SC    := fb_mem.STS.Resetting_SC,
										Holding_SC      := fb_mem.STS.Holding_SC,
										Unholding_SC    := fb_mem.STS.Unholding_SC,
										Suspending_SC   := fb_mem.STS.Suspending_SC,
										Unsuspending_SC := fb_mem.STS.Unsuspending_SC,
										Aborting_SC     := fb_mem.STS.Aborting_SC,
										Clearing_SC     := fb_mem.STS.Clearing_SC,
										Stopping_SC     := fb_mem.STS.Stopping_SC);

//********************************ZEROING***********************************								
fb_mem.STS.Starting_SC 		:= FALSE;
fb_mem.STS.Execute_SC 		:= FALSE;
fb_mem.STS.Resetting_SC 	:= FALSE;
fb_mem.STS.Holding_SC 		:= FALSE;
fb_mem.STS.Unholding_SC 	:= FALSE;
fb_mem.STS.Suspending_SC 	:= FALSE;
fb_mem.STS.Unsuspending_SC 	:= FALSE;
fb_mem.STS.Aborting_SC 		:= FALSE;
fb_mem.STS.Clearing_SC 		:= FALSE;
fb_mem.STS.Stopping_SC 		:= FALSE;
fb_mem.STS.Completing_SC 	:= FALSE;

//********************************init Modules***********************************
// Custom logic
EM_Can_Supply();
CM_Outfeed_ProductionLineSensor();

// Greyboxes
EM_Filling();
EM_CheckWeigher();
EM_BottomSeal();
EM_Labeller();
EM_TurningDevice();
EM_StampUnit();
EM_SealShrink();

// Transports
EM_Infeed_CheckWeigher();
EM_Transport_Checkweigher_BottomSeal();
EM_Transport_BottomSeal_Labeller();
EM_Transport_TurningDevice_StampUnit();
EM_Transport_StampUnit_SealShrink();

// Management logic
AlarmHandler();
ModeSelect();
//********************************TAGS instellen***********************************
//EM_Can_Supply
//CM_Outfeed_ProductionLineSensor.Tag := 'Outfeed production line Sensor';

EM_Filling();
EM_CheckWeigher();
EM_BottomSeal();
EM_Labeller();
EM_TurningDevice();
EM_StampUnit();
EM_SealShrink();
EM_Infeed_CheckWeigher();
EM_Transport_Checkweigher_BottomSeal();
EM_Transport_BottomSeal_Labeller();
EM_Transport_TurningDevice_StampUnit();
EM_Transport_StampUnit_SealShrink();

//********************************Auto manual logic***********************************
IF NOT bFirstCycleExecuted THEN
	EM_Can_Supply.Auto();
	//CM_Outfeed_ProductionLineSensor.Auto();
	EM_Filling.Auto();
	EM_CheckWeigher.Auto();
	EM_BottomSeal.Auto();
	EM_Labeller.Auto();
	EM_TurningDevice.Auto();
	EM_StampUnit.Auto();
	EM_SealShrink.Auto();
	EM_Infeed_CheckWeigher.Auto();
	EM_Transport_Checkweigher_BottomSeal.Auto();
	EM_Transport_BottomSeal_Labeller.Auto();
	EM_Transport_TurningDevice_StampUnit.Auto();
	EM_Transport_StampUnit_SealShrink.Auto();	
	bFirstCycleExecuted := TRUE;
END_IF

IF fb_mem.CS.Auto OR fb_mem.HMI.Auto THEN
	fb_mem.STS.Auto := TRUE;
	fb_mem.STS.Manueel := FALSE;
END_IF

IF fb_mem.CS.Manueel OR fb_mem.HMI.Manueel THEN
	fb_mem.STS.Auto := FALSE;
	fb_mem.STS.Manueel := TRUE;
END_IF

//********************************Control signals***********************************

IF fb_mem.CS.Reset THEN
	EM_Can_Supply.Reset();
//	CM_Outfeed_ProductionLineSensor.Reset();
	EM_Filling.Reset();
	EM_CheckWeigher.Reset();
	EM_BottomSeal.Reset();
	EM_Labeller.Reset();
	EM_TurningDevice.Reset();
	EM_StampUnit.Reset();
	EM_SealShrink.Reset();
	EM_Infeed_CheckWeigher.Reset();
	EM_Transport_Checkweigher_BottomSeal.Reset();
	EM_Transport_BottomSeal_Labeller.Reset();
	EM_Transport_TurningDevice_StampUnit.Reset();
	EM_Transport_StampUnit_SealShrink.Reset();
END_IF

IF fb_mem.CS.Abort THEN
	EM_Can_Supply.Abort();
//	CM_Outfeed_ProductionLineSensor.Abort();
	EM_Filling.Abort();
	EM_CheckWeigher.Abort();
	EM_BottomSeal.Abort();
	EM_Labeller.Abort();
	EM_TurningDevice.Abort();
	EM_StampUnit.Abort();
	EM_SealShrink.Abort();
	EM_Infeed_CheckWeigher.Abort();
	EM_Transport_Checkweigher_BottomSeal.Abort();
	EM_Transport_BottomSeal_Labeller.Abort();
	EM_Transport_TurningDevice_StampUnit.Abort();
	EM_Transport_StampUnit_SealShrink.Abort();
END_IF

IF fb_mem.CS.Clear THEN
	EM_Can_Supply.Clear();
//	CM_Outfeed_ProductionLineSensor.Clear();
	EM_Filling.Clear();
	EM_CheckWeigher.Clear();
	EM_BottomSeal.Clear();
	EM_Labeller.Clear();
	EM_TurningDevice.Clear();
	EM_StampUnit.Clear();
	EM_SealShrink.Clear();
	EM_Infeed_CheckWeigher.Clear();
	EM_Transport_Checkweigher_BottomSeal.Clear();
	EM_Transport_BottomSeal_Labeller.Clear();
	EM_Transport_TurningDevice_StampUnit.Clear();
	EM_Transport_StampUnit_SealShrink.Clear();
END_IF

IF fb_mem.CS.UnSuspend THEN
	EM_Can_Supply.UnSuspend();
//	CM_Outfeed_ProductionLineSensor.UnSuspend();
	EM_Filling.UnSuspend();
	EM_CheckWeigher.UnSuspend();
	EM_BottomSeal.UnSuspend();
	EM_Labeller.UnSuspend();
	EM_TurningDevice.UnSuspend();
	EM_StampUnit.UnSuspend();
	EM_SealShrink.UnSuspend();
	EM_Infeed_CheckWeigher.UnSuspend();
	EM_Transport_Checkweigher_BottomSeal.UnSuspend();
	EM_Transport_BottomSeal_Labeller.UnSuspend();
	EM_Transport_TurningDevice_StampUnit.UnSuspend();
	EM_Transport_StampUnit_SealShrink.UnSuspend();
END_IF

IF fb_mem.CS.Suspend THEN
	EM_Can_Supply.Suspend();
//	CM_Outfeed_ProductionLineSensor.Suspend();
	EM_Filling.Suspend();
	EM_CheckWeigher.Suspend();
	EM_BottomSeal.Suspend();
	EM_Labeller.Suspend();
	EM_TurningDevice.Suspend();
	EM_StampUnit.Suspend();
	EM_SealShrink.Suspend();
	EM_Infeed_CheckWeigher.Suspend();
	EM_Transport_Checkweigher_BottomSeal.Suspend();
	EM_Transport_BottomSeal_Labeller.Suspend();
	EM_Transport_TurningDevice_StampUnit.Suspend();
	EM_Transport_StampUnit_SealShrink.Suspend();
END_IF

IF fb_mem.CS.UnHold THEN
	EM_Can_Supply.UnHold();
//	CM_Outfeed_ProductionLineSensor.UnHold();
	EM_Filling.UnHold();
	EM_CheckWeigher.UnHold();
	EM_BottomSeal.UnHold();
	EM_Labeller.UnHold();
	EM_TurningDevice.UnHold();
	EM_StampUnit.UnHold();
	EM_SealShrink.UnHold();
	EM_Infeed_CheckWeigher.UnHold();
	EM_Transport_Checkweigher_BottomSeal.UnHold();
	EM_Transport_BottomSeal_Labeller.UnHold();
	EM_Transport_TurningDevice_StampUnit.UnHold();
	EM_Transport_StampUnit_SealShrink.UnHold();
END_IF

IF fb_mem.CS.Hold THEN
	EM_Can_Supply.Hold();
//	CM_Outfeed_ProductionLineSensor.Hold();
	EM_Filling.Hold();
	EM_CheckWeigher.Hold();
	EM_BottomSeal.Hold();
	EM_Labeller.Hold();
	EM_TurningDevice.Hold();
	EM_StampUnit.Hold();
	EM_SealShrink.Hold();
	EM_Infeed_CheckWeigher.Hold();
	EM_Transport_Checkweigher_BottomSeal.Hold();
	EM_Transport_BottomSeal_Labeller.Hold();
	EM_Transport_TurningDevice_StampUnit.Hold();
	EM_Transport_StampUnit_SealShrink.Hold();
END_IF

//*************Simulating SC statusses for the blackboxes********************
IF fb_mem.SIM.Starting_SC THEN
	EM_Can_Supply.Starting_SC();
	EM_Filling.Starting_SC();
	EM_CheckWeigher.Starting_SC();
	EM_BottomSeal.Starting_SC();
	EM_Labeller.Starting_SC();
	EM_StampUnit.Starting_SC();
	EM_SealShrink.Starting_SC();
	EM_TurningDevice.Starting_SC();
	EM_Infeed_CheckWeigher.Starting_SC();
	EM_Transport_Checkweigher_BottomSeal.Starting_SC();
	EM_Transport_BottomSeal_Labeller.Starting_SC();
	EM_Transport_TurningDevice_StampUnit.Starting_SC();
	EM_Transport_StampUnit_SealShrink.Starting_SC();
END_IF;
IF fb_mem.SIM.Execute_SC THEN
	fb_mem.STS.Execute_SC := TRUE;
	EM_Can_Supply.Execute_SC();
	EM_Filling.Execute_SC();
	EM_CheckWeigher.Execute_SC();
	EM_BottomSeal.Execute_SC();
	EM_Labeller.Execute_SC();
	EM_StampUnit.Execute_SC();
	EM_SealShrink.Execute_SC();
	EM_TurningDevice.Execute_SC();
	EM_Infeed_CheckWeigher.Execute_SC();
	EM_Transport_Checkweigher_BottomSeal.Execute_SC();
	EM_Transport_BottomSeal_Labeller.Execute_SC();
	EM_Transport_TurningDevice_StampUnit.Execute_SC();
	EM_Transport_StampUnit_SealShrink.Execute_SC();
END_IF;
IF fb_mem.SIM.Resetting_SC THEN
	EM_Can_Supply.Resetting_SC();
	EM_Filling.Resetting_SC();
	EM_CheckWeigher.Resetting_SC();
	EM_BottomSeal.Resetting_SC();
	EM_Labeller.Resetting_SC();
	EM_StampUnit.Resetting_SC();
	EM_SealShrink.Resetting_SC();
	EM_TurningDevice.Resetting_SC();
	EM_Infeed_CheckWeigher.Resetting_SC();
	EM_Transport_Checkweigher_BottomSeal.Resetting_SC();
	EM_Transport_BottomSeal_Labeller.Resetting_SC();
	EM_Transport_TurningDevice_StampUnit.Resetting_SC();
	EM_Transport_StampUnit_SealShrink.Resetting_SC();
END_IF;
IF fb_mem.SIM.Holding_SC THEN
	EM_Can_Supply.Holding_SC();
	EM_Filling.Holding_SC();
	EM_CheckWeigher.Holding_SC();
	EM_BottomSeal.Holding_SC();
	EM_Labeller.Holding_SC();
	EM_StampUnit.Holding_SC();
	EM_SealShrink.Holding_SC();
	EM_TurningDevice.Holding_SC();
	EM_Infeed_CheckWeigher.Holding_SC();
	EM_Transport_Checkweigher_BottomSeal.Holding_SC();
	EM_Transport_BottomSeal_Labeller.Holding_SC();
	EM_Transport_TurningDevice_StampUnit.Holding_SC();
	EM_Transport_StampUnit_SealShrink.Holding_SC();
END_IF;
IF fb_mem.SIM.Unholding_SC THEN
	EM_Can_Supply.Unholding_SC();
	EM_Filling.Unholding_SC();
	EM_CheckWeigher.Unholding_SC();
	EM_BottomSeal.Unholding_SC();
	EM_Labeller.Unholding_SC();
	EM_StampUnit.Unholding_SC();
	EM_SealShrink.Unholding_SC();
	EM_TurningDevice.Unholding_SC();
	EM_Infeed_CheckWeigher.Unholding_SC();
	EM_Transport_Checkweigher_BottomSeal.Unholding_SC();
	EM_Transport_BottomSeal_Labeller.Unholding_SC();
	EM_Transport_TurningDevice_StampUnit.Unholding_SC();
	EM_Transport_StampUnit_SealShrink.Unholding_SC();
END_IF;
IF fb_mem.SIM.Suspending_SC THEN
	EM_Can_Supply.Suspending_SC();
	EM_Filling.Suspending_SC();
	EM_CheckWeigher.Suspending_SC();
	EM_BottomSeal.Suspending_SC();
	EM_Labeller.Suspending_SC();
	EM_StampUnit.Suspending_SC();
	EM_SealShrink.Suspending_SC();
	EM_TurningDevice.Suspending_SC();
	EM_Infeed_CheckWeigher.Suspending_SC();
	EM_Transport_Checkweigher_BottomSeal.Suspending_SC();
	EM_Transport_BottomSeal_Labeller.Suspending_SC();
	EM_Transport_TurningDevice_StampUnit.Suspending_SC();
	EM_Transport_StampUnit_SealShrink.Suspending_SC();
END_IF;
IF fb_mem.SIM.Unsuspending_SC THEN
	EM_Can_Supply.Unsuspending_SC();
	EM_Filling.Unsuspending_SC();
	EM_CheckWeigher.Unsuspending_SC();
	EM_BottomSeal.Unsuspending_SC();
	EM_Labeller.Unsuspending_SC();
	EM_StampUnit.Unsuspending_SC();
	EM_SealShrink.Unsuspending_SC();
	EM_TurningDevice.Unsuspending_SC();
	EM_Infeed_CheckWeigher.Unsuspending_SC();
	EM_Transport_Checkweigher_BottomSeal.Unsuspending_SC();
	EM_Transport_BottomSeal_Labeller.Unsuspending_SC();
	EM_Transport_TurningDevice_StampUnit.Unsuspending_SC();
	EM_Transport_StampUnit_SealShrink.Unsuspending_SC();
END_IF;
IF fb_mem.SIM.Aborting_SC THEN
	fb_mem.STS.Aborting_SC := TRUE;
	EM_Can_Supply.Aborting_SC();
	EM_Filling.Aborting_SC();
	EM_CheckWeigher.Aborting_SC();
	EM_BottomSeal.Aborting_SC();
	EM_Labeller.Aborting_SC();
	EM_StampUnit.Aborting_SC();
	EM_SealShrink.Aborting_SC();
	EM_TurningDevice.Aborting_SC();
	EM_Infeed_CheckWeigher.Aborting_SC();
	EM_Transport_Checkweigher_BottomSeal.Aborting_SC();
	EM_Transport_BottomSeal_Labeller.Aborting_SC();
	EM_Transport_TurningDevice_StampUnit.Aborting_SC();
	EM_Transport_StampUnit_SealShrink.Aborting_SC();
END_IF;
IF fb_mem.SIM.Clearing_SC THEN
	EM_Can_Supply.Clearing_SC();
	EM_Filling.Clearing_SC();
	EM_CheckWeigher.Clearing_SC();
	EM_BottomSeal.Clearing_SC();
	EM_Labeller.Clearing_SC();
	EM_StampUnit.Clearing_SC();
	EM_SealShrink.Clearing_SC();
	EM_TurningDevice.Clearing_SC();
	EM_Infeed_CheckWeigher.Clearing_SC();
	EM_Transport_Checkweigher_BottomSeal.Clearing_SC();
	EM_Transport_BottomSeal_Labeller.Clearing_SC();
	EM_Transport_TurningDevice_StampUnit.Clearing_SC();
	EM_Transport_StampUnit_SealShrink.Clearing_SC();
END_IF;
IF fb_mem.SIM.Stopping_SC THEN
	EM_Can_Supply.Stopping_SC();
	EM_Filling.Stopping_SC();
	EM_CheckWeigher.Stopping_SC();
	EM_BottomSeal.Stopping_SC();
	EM_Labeller.Stopping_SC();
	EM_StampUnit.Stopping_SC();
	EM_SealShrink.Stopping_SC();
	EM_TurningDevice.Stopping_SC();
	EM_Infeed_CheckWeigher.Stopping_SC();
	EM_Transport_Checkweigher_BottomSeal.Stopping_SC();
	EM_Transport_BottomSeal_Labeller.Stopping_SC();
	EM_Transport_TurningDevice_StampUnit.Stopping_SC();
	EM_Transport_StampUnit_SealShrink.Stopping_SC();
END_IF

//********************************Exeptionhandling***********************************
// Puts line in HOLDING if a module is SUSPENDING
IF 	EM_Can_Supply.State 							= E_State_PackML.HOLDING OR
		EM_Filling.State 							= E_State_PackML.HOLDING OR
		EM_Infeed_CheckWeigher.State				= E_State_PackML.HOLDING OR
		EM_CheckWeigher.State 						= E_State_PackML.HOLDING OR
		EM_Transport_Checkweigher_BottomSeal.State	= E_State_PackML.HOLDING OR
		EM_BottomSeal.State							= E_State_PackML.HOLDING OR
		EM_Transport_BottomSeal_Labeller.State		= E_State_PackML.HOLDING OR
		EM_Labeller.State 							= E_State_PackML.HOLDING OR
		EM_TurningDevice.State						= E_State_PackML.HOLDING OR
		EM_Transport_TurningDevice_StampUnit.State	= E_State_PackML.HOLDING OR
		EM_StampUnit.State							= E_State_PackML.HOLDING OR
		EM_Transport_StampUnit_SealShrink.State		= E_State_PackML.HOLDING OR
		EM_SealShrink.State 						= E_State_PackML.HOLDING THEN
	fb_mem.CS.Suspend := TRUE;
	EM_Can_Supply.Suspend();
	EM_Filling.Suspend();
	EM_Infeed_CheckWeigher.Suspend();
	EM_CheckWeigher.Suspend();
	EM_Transport_Checkweigher_BottomSeal.Suspend();
	EM_BottomSeal.Suspend();
	EM_Transport_BottomSeal_Labeller.Suspend();
	EM_Labeller.Suspend();
	EM_TurningDevice.Suspend();
	EM_Transport_TurningDevice_StampUnit.Suspend();
	EM_StampUnit.Suspend();
	EM_Transport_StampUnit_SealShrink.Suspend();
	EM_SealShrink.Suspend();
END_IF

//********************************Action case***********************************
CASE fb_mem.STS.State OF
	E_State_PackML.IDLE 			: 
		IF fb_mem.CS.Start AND fb_mem.STS.Auto OR fb_mem.HMI.Start AND fb_mem.STS.Manueel THEN
		//do nothing
		END_IF
	
	E_State_PackML.STARTING 		:
		EM_Can_Supply.Start();
		IF EM_Can_Supply.State = E_State_PackML.EXECUTE THEN
			EM_Filling.Start();
			EM_Filling.Starting_SC();
			IF EM_Filling.State = E_State_PackML.EXECUTE THEN
				EM_Infeed_Checkweigher.Start();
				IF EM_Infeed_Checkweigher.State = E_State_PackML.EXECUTE THEN
					EM_CheckWeigher.Start();
					IF EM_CheckWeigher.State = E_State_PackML.EXECUTE THEN
						EM_Transport_CheckWeigher_BottomSeal.Start();
						IF EM_Transport_CheckWeigher_BottomSeal.State = E_State_PackML.EXECUTE THEN
							EM_BottomSeal.Start();
							IF EM_BottomSeal.State = E_State_PackML.EXECUTE THEN
								EM_Transport_BottomSeal_Labeller.Start();
								IF EM_Transport_BottomSeal_Labeller.State = E_State_PackML.EXECUTE THEN
									EM_Labeller.Start();
									IF EM_Labeller.State = E_State_PackML.EXECUTE THEN
										EM_TurningDevice.Start();
										IF EM_TurningDevice.State = E_State_PackML.EXECUTE THEN
											EM_Transport_TurningDevice_StampUnit.Start();
											IF EM_Transport_TurningDevice_StampUnit.State = E_State_PackML.EXECUTE THEN
												EM_Stampunit.Start();
												IF EM_Stampunit.State = E_State_PackML.EXECUTE THEN
													EM_Transport_StampUnit_SealShrink.Start();
													IF EM_Transport_StampUnit_SealShrink.State = E_State_PackML.EXECUTE THEN
														EM_SealShrink.Start();
														IF EM_SealShrink.State = E_State_PackML.EXECUTE THEN
															fb_mem.STS.Starting_SC := TRUE;
														END_IF;
													END_IF
												END_IF
											END_IF
										END_IF
									END_IF
								END_IF
							END_IF
						END_IF
					END_IF
				END_IF
			END_IF
		END_IF
	
	E_State_PackML.EXECUTE 			: 
		IF 	EM_Can_Supply.State 						= E_State_PackML.COMPLETE AND
			EM_Filling.State 							= E_State_PackML.COMPLETE AND
			EM_Infeed_CheckWeigher.State 				= E_State_PackML.COMPLETE AND
			EM_CheckWeigher.State 						= E_State_PackML.COMPLETE AND
			EM_Transport_Checkweigher_BottomSeal.State 	= E_State_PackML.COMPLETE AND
			EM_BottomSeal.State 						= E_State_PackML.COMPLETE AND
			EM_Transport_BottomSeal_Labeller.State 		= E_State_PackML.COMPLETE AND
			EM_Labeller.State 							= E_State_PackML.COMPLETE AND
			EM_TurningDevice.State 						= E_State_PackML.COMPLETE AND
			EM_Transport_TurningDevice_StampUnit.State 	= E_State_PackML.COMPLETE AND
			EM_StampUnit.State 							= E_State_PackML.COMPLETE AND
			EM_Transport_StampUnit_SealShrink.State 	= E_State_PackML.COMPLETE AND
			EM_SealShrink.State 						= E_State_PackML.COMPLETE THEN
		fb_mem.STS.Execute_SC := TRUE;
		END_IF
	E_State_PackML.COMPLETING 		:
		IF 	EM_Can_Supply.State 						= E_State_PackML.COMPLETE AND
			EM_Filling.State 							= E_State_PackML.COMPLETE AND
			EM_Infeed_CheckWeigher.State				= E_State_PackML.COMPLETE AND
			EM_CheckWeigher.State 						= E_State_PackML.COMPLETE AND
			EM_Transport_Checkweigher_BottomSeal.State	= E_State_PackML.COMPLETE AND
			EM_BottomSeal.State							= E_State_PackML.COMPLETE AND
			EM_Transport_BottomSeal_Labeller.State		= E_State_PackML.COMPLETE AND
			EM_Labeller.State 							= E_State_PackML.COMPLETE AND
			EM_TurningDevice.State						= E_State_PackML.COMPLETE AND
			EM_Transport_TurningDevice_StampUnit.State	= E_State_PackML.COMPLETE AND
			EM_StampUnit.State							= E_State_PackML.COMPLETE AND
			EM_Transport_StampUnit_SealShrink.State		= E_State_PackML.COMPLETE AND
			EM_SealShrink.State 						= E_State_PackML.COMPLETE THEN
		fb_mem.STS.Completing_SC := TRUE;
		END_IF
	E_State_PackML.COMPLETE 		:
		IF fb_mem.CS.Clear AND fb_mem.STS.Auto OR fb_mem.HMI.Clear AND fb_mem.STS.Manueel THEN
			fb_mem.STS.Completing_SC := TRUE;
		END_IF
	
	E_State_PackML.RESETTING 		:
		IF 	EM_Can_Supply.State 						= E_State_PackML.IDLE AND
			EM_Filling.State 							= E_State_PackML.IDLE AND
			EM_Infeed_CheckWeigher.State				= E_State_PackML.IDLE AND
			EM_CheckWeigher.State 						= E_State_PackML.IDLE AND
			EM_Transport_Checkweigher_BottomSeal.State	= E_State_PackML.IDLE AND
			EM_BottomSeal.State							= E_State_PackML.IDLE AND
			EM_Transport_BottomSeal_Labeller.State		= E_State_PackML.IDLE AND
			EM_Labeller.State 							= E_State_PackML.IDLE AND
			EM_TurningDevice.State						= E_State_PackML.IDLE AND
			EM_Transport_TurningDevice_StampUnit.State	= E_State_PackML.IDLE AND
			EM_StampUnit.State							= E_State_PackML.IDLE AND
			EM_Transport_StampUnit_SealShrink.State		= E_State_PackML.IDLE AND
			EM_SealShrink.State 						= E_State_PackML.IDLE THEN
		//State complete:
		fb_mem.STS.Resetting_SC := TRUE;
		END_IF
	
	E_State_PackML.HOLDING 			:	// TO BE PROGRAMMED
		IF 	EM_Can_Supply.State 							= E_State_PackML.HELD AND
				EM_Filling.State 							= E_State_PackML.HELD AND
				EM_Infeed_CheckWeigher.State				= E_State_PackML.HELD AND
				EM_CheckWeigher.State 						= E_State_PackML.HELD AND
				EM_Transport_Checkweigher_BottomSeal.State	= E_State_PackML.HELD AND
				EM_BottomSeal.State							= E_State_PackML.HELD AND
				EM_Transport_BottomSeal_Labeller.State		= E_State_PackML.HELD AND
				EM_Labeller.State 							= E_State_PackML.HELD AND
				EM_TurningDevice.State						= E_State_PackML.HELD AND
				EM_Transport_TurningDevice_StampUnit.State	= E_State_PackML.HELD AND
				EM_StampUnit.State							= E_State_PackML.HELD AND
				EM_Transport_StampUnit_SealShrink.State		= E_State_PackML.HELD AND
				EM_SealShrink.State 						= E_State_PackML.HELD THEN
			fb_mem.STS.Holding_SC := TRUE;
		END_IF 
		
	
	E_State_PackML.HELD 			:	// TO BE PROGRAMMED
		//Not defined
	
	
	E_State_PackML.UNHOLDING 		:	
		IF 	EM_Can_Supply.State 							= E_State_PackML.EXECUTE AND
				EM_Filling.State 							= E_State_PackML.EXECUTE AND
				EM_Infeed_CheckWeigher.State				= E_State_PackML.EXECUTE AND
				EM_CheckWeigher.State 						= E_State_PackML.EXECUTE AND
				EM_Transport_Checkweigher_BottomSeal.State	= E_State_PackML.EXECUTE AND
				EM_BottomSeal.State							= E_State_PackML.EXECUTE AND
				EM_Transport_BottomSeal_Labeller.State		= E_State_PackML.EXECUTE AND
				EM_Labeller.State 							= E_State_PackML.EXECUTE AND
				EM_TurningDevice.State						= E_State_PackML.EXECUTE AND
				EM_Transport_TurningDevice_StampUnit.State	= E_State_PackML.EXECUTE AND
				EM_StampUnit.State							= E_State_PackML.EXECUTE AND
				EM_Transport_StampUnit_SealShrink.State		= E_State_PackML.EXECUTE AND
				EM_SealShrink.State 						= E_State_PackML.EXECUTE THEN
			fb_mem.STS.Unholding_SC := TRUE;
		END_IF 
	
	
	E_State_PackML.SUSPENDING 		:
		IF (EM_Can_Supply.State 						= E_State_PackML.SUSPENDED OR
			EM_Can_Supply.State 						= E_State_PackML.HELD) AND
		   (EM_Filling.State 							= E_State_PackML.SUSPENDED OR
			EM_Filling.State 							= E_State_PackML.HELD) AND
		   (EM_Infeed_CheckWeigher.State				= E_State_PackML.SUSPENDED OR
			EM_Infeed_CheckWeigher.State				= E_State_PackML.HELD) AND
		   (EM_CheckWeigher.State 						= E_State_PackML.SUSPENDED OR
			EM_CheckWeigher.State 						= E_State_PackML.HELD) AND
		   (EM_Transport_Checkweigher_BottomSeal.State	= E_State_PackML.SUSPENDED OR
			EM_Transport_Checkweigher_BottomSeal.State	= E_State_PackML.HELD) AND
		   (EM_BottomSeal.State							= E_State_PackML.SUSPENDED OR
			EM_BottomSeal.State 						= E_State_PackML.HELD) AND
		   (EM_Transport_BottomSeal_Labeller.State		= E_State_PackML.SUSPENDED OR
			EM_Transport_BottomSeal_Labeller.State 		= E_State_PackML.HELD) AND
		   (EM_Labeller.State 							= E_State_PackML.SUSPENDED OR
			EM_Labeller.State 							= E_State_PackML.HELD) AND
		   (EM_TurningDevice.State						= E_State_PackML.SUSPENDED OR
			EM_TurningDevice.State 						= E_State_PackML.HELD) AND
		   (EM_Transport_TurningDevice_StampUnit.State	= E_State_PackML.SUSPENDED OR
			EM_Transport_TurningDevice_StampUnit.State	= E_State_PackML.HELD) AND
		   (EM_StampUnit.State							= E_State_PackML.SUSPENDED OR
			EM_StampUnit.State							= E_State_PackML.HELD) AND
		   (EM_Transport_StampUnit_SealShrink.State		= E_State_PackML.SUSPENDED OR
			EM_Transport_StampUnit_SealShrink.State		= E_State_PackML.HELD) AND
		   (EM_SealShrink.State 						= E_State_PackML.SUSPENDED OR 
			EM_SealShrink.State							= E_State_PackML.HELD) THEN
		fb_mem.STS.Suspending_SC := TRUE;
		END_IF
	
	E_State_PackML.SUSPENDED 		:
		IF	EM_Can_Supply.State 						= E_State_PackML.UNHOLDING OR
			EM_Filling.State 							= E_State_PackML.UNHOLDING OR
			EM_Infeed_CheckWeigher.State				= E_State_PackML.UNHOLDING OR
			EM_CheckWeigher.State 						= E_State_PackML.UNHOLDING OR
			EM_Transport_Checkweigher_BottomSeal.State	= E_State_PackML.UNHOLDING OR
			EM_BottomSeal.State							= E_State_PackML.UNHOLDING OR
			EM_Transport_BottomSeal_Labeller.State		= E_State_PackML.UNHOLDING OR
			EM_Labeller.State 							= E_State_PackML.UNHOLDING OR
			EM_TurningDevice.State						= E_State_PackML.UNHOLDING OR
			EM_Transport_TurningDevice_StampUnit.State	= E_State_PackML.UNHOLDING OR
			EM_StampUnit.State							= E_State_PackML.UNHOLDING OR
			EM_Transport_StampUnit_SealShrink.State		= E_State_PackML.UNHOLDING OR
			EM_SealShrink.State 						= E_State_PackML.UNHOLDING THEN 
		fb_mem.CS.Unsuspend := TRUE;
		EM_Can_Supply.Unsuspend();
		EM_Filling.Unsuspend();
		EM_Infeed_CheckWeigher.Start();
		EM_CheckWeigher.Unsuspend();
		EM_Transport_Checkweigher_BottomSeal.Start();
		EM_BottomSeal.Unsuspend();
		EM_Transport_BottomSeal_Labeller.Start();
		EM_Labeller.Unsuspend();
		EM_TurningDevice.Unsuspend();
		EM_Transport_TurningDevice_StampUnit.Start();
		EM_StampUnit.Unsuspend();
		EM_Transport_StampUnit_SealShrink.Start();
		EM_SealShrink.Unsuspend();
		END_IF
	
	E_State_PackML.UNSUSPENDING 	:
		fb_mem.STS.Unsuspending_SC	:= TRUE;
	
	E_State_PackML.ABORTING			:
		IF 	EM_Can_Supply.State 							= E_State_PackML.ABORTED AND
				EM_Filling.State 							= E_State_PackML.ABORTED AND
				EM_Infeed_CheckWeigher.State				= E_State_PackML.ABORTED AND
				EM_CheckWeigher.State 						= E_State_PackML.ABORTED AND
				EM_Transport_Checkweigher_BottomSeal.State	= E_State_PackML.ABORTED AND
				EM_BottomSeal.State							= E_State_PackML.ABORTED AND
				EM_Transport_BottomSeal_Labeller.State		= E_State_PackML.ABORTED AND
				EM_Labeller.State 							= E_State_PackML.ABORTED AND
				EM_TurningDevice.State						= E_State_PackML.ABORTED AND
				EM_Transport_TurningDevice_StampUnit.State	= E_State_PackML.ABORTED AND
				EM_StampUnit.State							= E_State_PackML.ABORTED AND
				EM_Transport_StampUnit_SealShrink.State		= E_State_PackML.ABORTED AND
				EM_SealShrink.State 						= E_State_PackML.ABORTED THEN
			fb_mem.STS.Aborting_SC := TRUE;
		END_IF
	
	E_State_PackML.ABORTED			:
		IF fb_mem.CS.Clear AND fb_mem.STS.Auto OR fb_mem.HMI.Clear AND fb_mem.STS.Manueel THEN
			fb_mem.CS.Clear 							:= TRUE;
			EM_Can_Supply.Clear();
			EM_Filling.Clear();
			EM_Infeed_CheckWeigher.Clear();
			EM_CheckWeigher.Clear();
			EM_Transport_Checkweigher_BottomSeal.Clear();
			EM_BottomSeal.Clear();
			EM_Transport_BottomSeal_Labeller.Clear();
			EM_Labeller.Clear();
			EM_TurningDevice.Clear();
			EM_Transport_TurningDevice_StampUnit.Clear();
			EM_StampUnit.Clear();
			EM_Transport_StampUnit_SealShrink.Clear();
			EM_SealShrink.Clear();
		END_IF
	
	E_State_PackML.CLEARING 		:
		IF 	EM_Can_Supply.State 							= E_State_PackML.STOPPED AND
				EM_Filling.State 							= E_State_PackML.STOPPED AND
				EM_Infeed_CheckWeigher.State				= E_State_PackML.STOPPED AND
				EM_CheckWeigher.State 						= E_State_PackML.STOPPED AND
				EM_Transport_Checkweigher_BottomSeal.State	= E_State_PackML.STOPPED AND
				EM_BottomSeal.State							= E_State_PackML.STOPPED AND
				EM_Transport_BottomSeal_Labeller.State		= E_State_PackML.STOPPED AND
				EM_Labeller.State 							= E_State_PackML.STOPPED AND
				EM_TurningDevice.State						= E_State_PackML.STOPPED AND
				EM_Transport_TurningDevice_StampUnit.State	= E_State_PackML.STOPPED AND
				EM_StampUnit.State							= E_State_PackML.STOPPED AND
				EM_Transport_StampUnit_SealShrink.State		= E_State_PackML.STOPPED AND
				EM_SealShrink.State 						= E_State_PackML.STOPPED THEN
			fb_mem.STS.Clearing_SC := TRUE;
		END_IF
	
	E_State_PackML.STOPPING 		:
		EM_Can_Supply.Stop();
		EM_Filling.Stop();
		EM_Infeed_CheckWeigher.Stop();
		EM_CheckWeigher.Stop();
		EM_Transport_Checkweigher_BottomSeal.Stop();
		EM_BottomSeal.Stop();
		EM_Transport_BottomSeal_Labeller.Stop();
		EM_Labeller.Stop();
		EM_TurningDevice.Stop();
		EM_Transport_TurningDevice_StampUnit.Stop();
		EM_StampUnit.Stop();
		EM_Transport_StampUnit_SealShrink.Stop();
		EM_SealShrink.Stop();
		IF 	EM_Can_Supply.State 							= E_State_PackML.STOPPED AND
				EM_Filling.State 							= E_State_PackML.STOPPED AND
				EM_Infeed_CheckWeigher.State				= E_State_PackML.STOPPED AND
				EM_CheckWeigher.State 						= E_State_PackML.STOPPED AND
				EM_Transport_Checkweigher_BottomSeal.State	= E_State_PackML.STOPPED AND
				EM_BottomSeal.State							= E_State_PackML.STOPPED AND
				EM_Transport_BottomSeal_Labeller.State		= E_State_PackML.STOPPED AND
				EM_Labeller.State 							= E_State_PackML.STOPPED AND
				EM_TurningDevice.State						= E_State_PackML.STOPPED AND
				EM_Transport_TurningDevice_StampUnit.State	= E_State_PackML.STOPPED AND
				EM_StampUnit.State							= E_State_PackML.STOPPED AND
				EM_Transport_StampUnit_SealShrink.State		= E_State_PackML.STOPPED AND
				EM_SealShrink.State 						= E_State_PackML.STOPPED THEN
			fb_mem.STS.Stopping_SC := TRUE;
		END_IF 
	
	E_State_PackML.STOPPED 			:
		IF (fb_mem.CS.Reset AND fb_mem.STS.Auto) OR (fb_mem.HMI.Reset AND fb_mem.STS.Manueel) THEN
			fb_mem.CS.Reset := TRUE;
			EM_Can_Supply.Reset();
			EM_Filling.Reset();
			EM_Infeed_CheckWeigher.Reset();
			EM_CheckWeigher.Reset();
			EM_Transport_Checkweigher_BottomSeal.Reset();
			EM_BottomSeal.Reset();
			EM_Transport_BottomSeal_Labeller.Reset();
			EM_Labeller.Reset();
			EM_TurningDevice.Reset();
			EM_Transport_TurningDevice_StampUnit.Reset();
			EM_StampUnit.Reset();
			EM_Transport_StampUnit_SealShrink.Reset();
			EM_SealShrink.Reset();
		END_IF 
	ELSE
		fb_mem.STS.State := E_State_PackML.SUSPENDING;
END_CASE

//********************************HMI_Connection***********************************
fb_mem.STS.StringState     := TO_STRING(fb_mem.STS.State);

//********************************ZEROING***********************************

fb_mem.CS.Auto            := FALSE;
fb_mem.CS.Manueel         := FALSE;
fb_mem.CS.Start           := FALSE;
fb_mem.CS.Stop            := FALSE;
fb_mem.CS.Reset           := FALSE;
fb_mem.CS.Abort           := FALSE;
fb_mem.CS.Clear           := FALSE;
fb_mem.CS.UnSuspend       := FALSE;
fb_mem.CS.Suspend         := FALSE;
fb_mem.CS.UnHold          := FALSE;
fb_mem.CS.Hold            := FALSE;


fb_mem.HMI.Auto            := FALSE;
fb_mem.HMI.Manueel         := FALSE;
fb_mem.HMI.Start           := FALSE;
fb_mem.HMI.Stop            := FALSE;
fb_mem.HMI.Reset           := FALSE;
fb_mem.HMI.Abort           := FALSE;
fb_mem.HMI.Clear           := FALSE;
fb_mem.HMI.UnSuspend       := FALSE;
fb_mem.HMI.Suspend         := FALSE;
fb_mem.HMI.UnHold          := FALSE;
fb_mem.HMI.Hold            := FALSE;

{warning 'add method implementation '}
METHOD Abort : BOOL
fb_mem.CS.Abort := TRUE;
END_METHOD

{warning 'add method implementation '}
METHOD Auto : BOOL
fb_mem.CS.Auto := TRUE;
Auto := fb_mem.STS.Auto;
END_METHOD

{warning 'add method implementation '}
METHOD Clear : BOOL
fb_mem.CS.Clear := TRUE;
END_METHOD

METHOD FB_init : BOOL
VAR_INPUT
	bInitRetains : BOOL; // if TRUE, the retain variables are initialized (warm start / cold start)
	bInCopyCode : BOOL;  // if TRUE, the instance afterwards gets moved into the copy code (online change)
END_VAR
//**************************INITIATE**************************//
//Custom logic
EM_Can_Supply.FB_init(0,0);
EM_TurningDevice.FB_init(0,0);
CM_Outfeed_ProductionLineSensor.FB_init(0,0);
	
//PackML machine's
EM_Filling.FB_init(0,0);
EM_CheckWeigher.FB_init(0,0);
EM_BottomSeal.FB_init(0,0);
EM_Labeller.FB_init(0,0);
EM_TurningDevice.FB_init(0,0);
EM_StampUnit.FB_init(0,0);
EM_SealShrink.FB_init(0,0);
	
//Transport logic
EM_Infeed_CheckWeigher.FB_init(0,0);
EM_Transport_Checkweigher_BottomSeal.FB_init(0,0);
EM_Transport_BottomSeal_Labeller.FB_init(0,0);
EM_Transport_TurningDevice_StampUnit.FB_init(0,0);
EM_Transport_StampUnit_SealShrink.FB_init(0,0);
END_METHOD

{warning 'add method implementation '}
METHOD Hold : BOOL
fb_mem.CS.Hold := TRUE;
END_METHOD

{warning 'add method implementation '}
METHOD Manueel : BOOL
fb_mem.CS.Manueel := TRUE;
Manueel := fb_mem.STS.Manueel;
END_METHOD

{warning 'add method implementation '}
METHOD Reset : BOOL
fb_mem.CS.Reset := TRUE;
END_METHOD

{warning 'add method implementation '}
METHOD Start : BOOL
fb_mem.CS.Start := TRUE;
END_METHOD

{warning 'add property implementation'}
PROPERTY State : E_State_PackML
GET
State := fb_mem.STS.State;
END_GET
END_PROPERTY

{warning 'add method implementation '}
METHOD Stop : BOOL
fb_mem.CS.Stop := TRUE;
END_METHOD

{warning 'add method implementation '}
METHOD Suspend : BOOL
fb_mem.CS.Suspend := TRUE;
END_METHOD

{warning 'add method implementation '}
METHOD Unhold : BOOL
fb_mem.CS.Unhold := TRUE;
END_METHOD

{warning 'add method implementation '}
METHOD Unsuspend : BOOL
fb_mem.CS.Unsuspend := TRUE;
END_METHOD

{warning 'add method implementation '}
METHOD ZeroAllVar : BOOL
END_METHOD

END_FUNCTION_BLOCK

// ---- POUs/2. Equipment Modules/1. EM_Can_Supply/EM_Can_Supply.TcPOU
FUNCTION_BLOCK EM_Can_Supply IMPLEMENTS ITF_Can_Supply, ITF_PackML
VAR
	fb_mem : STRUCT_EM_CanSupply;
	bFirstCycleExecuted : BOOL;
	
	//SubModules
	EM_Transport_Can_Supply1		: EM_Transport_Mechanische_Stop;
	EM_Transport_Can_Supply2		: EM_Transport;
	Sen_A1_Near						: CM_Sensor;
	Sen_A1_Far						: CM_Sensor;
	Sen_A2_Near						: CM_Sensor;
	Sen_A2_Far						: CM_Sensor;
	ValveDirection					: CM_Valve;  
END_VAR

(*
Tijn Verdurmen
*)//********************************Initiating***********************************
fb_mem.STS.State := PackML_StateMachine(State			:= fb_mem.STS.State,
										Start           := fb_mem.CS.Start,
										Stop            := fb_mem.CS.Stop,
										Reset           := fb_mem.CS.Reset,
										Abort           := fb_mem.CS.Abort,
										Clear           := fb_mem.CS.Clear,
										UnSuspend       := fb_mem.CS.UnSuspend,
										Suspend         := fb_mem.CS.Suspend,
										UnHold          := fb_mem.CS.UnHold,
										Hold            := fb_mem.CS.Hold,
										Starting_SC     := fb_mem.STS.Starting_SC,
										Execute_SC      := fb_mem.STS.Execute_SC,
										Completing_SC	:= fb_mem.STS.Completing_SC,
										Resetting_SC    := fb_mem.STS.Resetting_SC,
										Holding_SC      := fb_mem.STS.Holding_SC,
										Unholding_SC    := fb_mem.STS.Unholding_SC,
										Suspending_SC   := fb_mem.STS.Suspending_SC,
										Unsuspending_SC := fb_mem.STS.Unsuspending_SC,
										Aborting_SC     := fb_mem.STS.Aborting_SC,
										Clearing_SC     := fb_mem.STS.Clearing_SC,
										Stopping_SC     := fb_mem.STS.Stopping_SC);

//********************************Init***********************************
EM_Transport_Can_Supply1();
EM_Transport_Can_Supply2();			
										
//********************************ZEROING***********************************								
fb_mem.STS.Starting_SC 		:= FALSE;
fb_mem.STS.Execute_SC 		:= FALSE;
fb_mem.STS.Resetting_SC 	:= FALSE;
fb_mem.STS.Holding_SC 		:= FALSE;
fb_mem.STS.Unholding_SC 	:= FALSE;
fb_mem.STS.Suspending_SC 	:= FALSE;
fb_mem.STS.Unsuspending_SC 	:= FALSE;
fb_mem.STS.Aborting_SC 		:= FALSE;
fb_mem.STS.Clearing_SC 		:= FALSE;
fb_mem.STS.Stopping_SC 		:= FALSE;
fb_mem.STS.Completing_SC 	:= FALSE;

//********************************Auto manual logic***********************************
IF NOT bFirstCycleExecuted THEN
	EM_Transport_Can_Supply1.Auto();
	EM_Transport_Can_Supply2.Auto();
	ValveDirection.Auto := TRUE;
	bFirstCycleExecuted := TRUE;
END_IF

IF fb_mem.CS.Auto OR fb_mem.HMI.Auto THEN
	fb_mem.STS.Auto := TRUE;
	fb_mem.STS.Manueel := FALSE;
END_IF

IF fb_mem.CS.Manueel OR fb_mem.HMI.Manueel THEN
	fb_mem.STS.Auto := FALSE;
	fb_mem.STS.Manueel := TRUE;
END_IF

//********************Manupilatie***********8
IF fb_mem.SIM.Sen_A1_Near_TRUE THEN
	Sen_A1_Near.Output := TRUE;
END_IF
IF fb_mem.SIM.Sen_A1_Far_TRUE THEN
	Sen_A1_Far.Output := TRUE;
END_IF
IF fb_mem.SIM.Sen_A2_Near_TRUE THEN
	Sen_A2_Near.Output := TRUE;
END_IF
IF fb_mem.SIM.Sen_A2_Far_TRUE THEN
	Sen_A2_Far.Output := TRUE;
END_IF

//********************************Exeptionhandling***********************************

//********************************Action case***********************************
CASE fb_mem.STS.State OF
	E_State_PackML.IDLE 			: 
		//Do nothing
	E_State_PackML.STARTING 		:
		EM_Transport_Can_Supply1.Start();
		EM_Transport_Can_Supply2.Start();
		IF ((EM_Transport_Can_Supply1.State= E_State_PackML.EXECUTE) AND (EM_Transport_Can_Supply2.State= E_State_PackML.EXECUTE)) THEN
			ValveDirection.Close();	//=naar filler 1
				IF Sen_A1_Far.Output=TRUE AND Sen_A1_Near.Output=TRUE THEN //filler 2 hoeft nog niet vol te zijn om te starten
					ValveDirection.Open();	//=naar filler 2
					fb_mem.STS.Starting_SC := TRUE;
				END_IF
		END_IF
		
	E_State_PackML.EXECUTE		: // dit was execute
		//Hier heen en weer swichen totdat bijden buffers vol zijn en dus alle sensoren waar zijn met filler 1 prioriteit
		//Als Sen_A1_Far AND Sen_A1_Near AND !Sen_A2_Near THEN wissel naar A2 en vise versa
		IF Sen_A1_Far.Output=TRUE AND Sen_A2_Far.Output=TRUE AND Sen_A1_Near.Output=TRUE AND Sen_A2_Near.Output=FALSE THEN
			ValveDirection.Open();	//Richting_L naar filler 2 heet open
		END_IF
		IF Sen_A1_Far.Output=TRUE AND Sen_A2_Far.Output=TRUE AND Sen_A2_Near.Output=TRUE AND Sen_A1_Near.Output=FALSE THEN
			ValveDirection.Close();	//Richting_L naar filler 1
		END_IF
		IF Sen_A1_Far.Output=FALSE THEN
			ValveDirection.Close();		//Richting_L naar filler 1 heet close
		END_IF
	E_State_PackML.COMPLETING		:
		EM_Transport_Can_Supply1.Execute_SC();
		EM_Transport_Can_Supply2.Execute_SC();
		IF EM_Transport_Can_Supply1.State = E_State_PackML.COMPLETE AND EM_Transport_Can_Supply2.State = E_State_PackML.COMPLETE THEN
			fb_mem.STS.Completing_SC := TRUE;
		END_IF
	E_State_PackML.COMPLETE 		:
		fb_mem.STS.Completing_SC:=TRUE;
		
	E_State_PackML.RESETTING 		:
		EM_Transport_Can_Supply1.Reset();
		EM_Transport_Can_Supply2.Reset();
		IF	((EM_Transport_Can_Supply1.State= E_State_PackML.IDLE) AND (EM_Transport_Can_Supply2.State= E_State_PackML.IDLE)) THEN
			fb_mem.STS.Resetting_SC:=TRUE;
		END_IF
		
	E_State_PackML.HOLDING 			:
		EM_Transport_Can_Supply1.Hold();
		EM_Transport_Can_Supply2.Hold();
		IF	((EM_Transport_Can_Supply1.State= E_State_PackML.HELD) AND (EM_Transport_Can_Supply2.State= E_State_PackML.HELD)) THEN
			fb_mem.STS.Holding_SC:=TRUE;
		END_IF
		
	E_State_PackML.HELD 			:
		// Do nothing
	E_State_PackML.UNHOLDING 		:
		EM_Transport_Can_Supply1.Unhold();
		EM_Transport_Can_Supply2.Unhold();
		IF	((EM_Transport_Can_Supply1.State= E_State_PackML.EXECUTE) AND (EM_Transport_Can_Supply2.State= E_State_PackML.EXECUTE)) THEN
			fb_mem.STS.Unholding_SC:=TRUE;
		END_IF
		
	E_State_PackML.SUSPENDING 		:
		EM_Transport_Can_Supply1.Suspend();
		EM_Transport_Can_Supply2.Suspend();
		IF	((EM_Transport_Can_Supply1.State= E_State_PackML.SUSPENDED) AND (EM_Transport_Can_Supply2.State= E_State_PackML.SUSPENDED)) THEN
			fb_mem.STS.Suspending_SC:=TRUE;
		END_IF
		
	E_State_PackML.SUSPENDED 		:
		// Do nothing
		
	E_State_PackML.UNSUSPENDING 	:
		EM_Transport_Can_Supply1.Unsuspend();
		EM_Transport_Can_Supply2.Unsuspend();
		IF	((EM_Transport_Can_Supply1.State= E_State_PackML.EXECUTE) AND (EM_Transport_Can_Supply2.State= E_State_PackML.EXECUTE)) THEN
			fb_mem.STS.Unsuspending_SC:=TRUE;
		END_IF
	
	E_State_PackML.ABORTING			:
		EM_Transport_Can_Supply1.Abort();
		EM_Transport_Can_Supply2.Abort();
		IF	((EM_Transport_Can_Supply1.State= E_State_PackML.ABORTED) AND (EM_Transport_Can_Supply2.State= E_State_PackML.ABORTED)) THEN
			fb_mem.STS.Aborting_SC:=TRUE;
		END_IF
		
	E_State_PackML.ABORTED			:
		// Do nothing
		
	E_State_PackML.CLEARING 		:
		EM_Transport_Can_Supply1.Clear();
		EM_Transport_Can_Supply2.Clear();
		IF	((EM_Transport_Can_Supply1.State= E_State_PackML.STOPPED) AND (EM_Transport_Can_Supply2.State= E_State_PackML.STOPPED)) THEN
			fb_mem.STS.Clearing_SC:=TRUE;
		END_IF
		
	E_State_PackML.STOPPED			:
		// DO nothing
END_CASE 
//********************************HMI_Connection***********************************
fb_mem.STS.StringState     := TO_STRING(fb_mem.STS.State); 

//********************************ZEROING***********************************

fb_mem.CS.Auto            := FALSE;
fb_mem.CS.Manueel         := FALSE;
fb_mem.CS.Start           := FALSE;
fb_mem.CS.Stop            := FALSE;
fb_mem.CS.Reset           := FALSE;
fb_mem.CS.Abort           := FALSE;
fb_mem.CS.Clear           := FALSE;
fb_mem.CS.UnSuspend       := FALSE;
fb_mem.CS.Suspend         := FALSE;
fb_mem.CS.UnHold          := FALSE;
fb_mem.CS.Hold            := FALSE;

{warning 'add method implementation '}
METHOD Abort : BOOL
fb_mem.CS.Abort := TRUE;
END_METHOD

METHOD Aborting_SC : BOOL
VAR_INPUT
END_VAR
fb_mem.STS.Aborting_SC := TRUE;
END_METHOD

{warning 'add method implementation '}
METHOD Auto : BOOL
fb_mem.CS.Auto := TRUE;
Auto := fb_mem.STS.Auto;
END_METHOD

{warning 'add method implementation '}
METHOD Clear : BOOL
fb_mem.CS.Clear := TRUE;
END_METHOD

METHOD Clearing_SC : BOOL
VAR_INPUT
END_VAR
fb_mem.STS.Clearing_SC := TRUE;
END_METHOD

METHOD Completing_SC : BOOL
VAR_INPUT
END_VAR
fb_mem.STS.Completing_SC := TRUE;
END_METHOD

METHOD Execute_SC : BOOL
VAR_INPUT
END_VAR
fb_mem.STS.Execute_SC := TRUE;
END_METHOD

{warning 'add method implementation '}
METHOD FB_init : BOOL
VAR_INPUT
	bInitRetains : BOOL; // if TRUE, the retain variables are initialized (warm start / cold start)
	bInCopyCode : BOOL;  // if TRUE, the instance afterwards gets moved into the copy code (online change)
END_VAR
END_METHOD

{warning 'add method implementation '}
METHOD Hold : BOOL
fb_mem.CS.Hold := TRUE;
END_METHOD

METHOD Holding_SC : BOOL
VAR_INPUT
END_VAR
fb_mem.STS.Holding_SC := TRUE;
END_METHOD

{warning 'add method implementation '}
METHOD Manueel : BOOL
fb_mem.CS.Manueel := TRUE;
Manueel := fb_mem.STS.Manueel;
END_METHOD

{warning 'add method implementation '}
METHOD Reset : BOOL
fb_mem.CS.Reset := TRUE;
END_METHOD

METHOD Resetting_SC : BOOL
VAR_INPUT
END_VAR
fb_mem.STS.Resetting_SC := TRUE;
END_METHOD

{warning 'add method implementation '}
METHOD Start : BOOL
fb_mem.CS.Start := TRUE;
END_METHOD

METHOD Starting_SC : BOOL
VAR_INPUT
END_VAR
fb_mem.STS.Starting_SC := TRUE;
END_METHOD

{warning 'add property implementation'}
PROPERTY State : E_State_PackML
GET
State := fb_mem.STS.State;
END_GET
END_PROPERTY

{warning 'add method implementation '}
METHOD Stop : BOOL
fb_mem.CS.Stop := TRUE;
END_METHOD

METHOD Stopping_SC : BOOL
VAR_INPUT
END_VAR
fb_mem.STS.Stopping_SC := TRUE;
END_METHOD

{warning 'add method implementation '}
METHOD Suspend : BOOL
fb_mem.CS.Suspend := TRUE;
END_METHOD

METHOD Suspending_SC : BOOL
VAR_INPUT
END_VAR
fb_mem.STS.Suspending_SC := TRUE;
END_METHOD

{warning 'add method implementation '}
METHOD Unhold : BOOL
fb_mem.CS.Unhold := TRUE;
END_METHOD

METHOD Unholding_SC : BOOL
VAR_INPUT
END_VAR
fb_mem.STS.Unholding_SC := TRUE;
END_METHOD

{warning 'add method implementation '}
METHOD Unsuspend : BOOL
fb_mem.CS.Unsuspend := TRUE;
END_METHOD

METHOD Unsuspending_SC : BOOL
VAR_INPUT
END_VAR
fb_mem.STS.Unsuspending_SC := TRUE;
END_METHOD

{warning 'add method implementation '}
METHOD ZeroAllVar : BOOL
END_METHOD

END_FUNCTION_BLOCK

// ---- POUs/2. Equipment Modules/5. EM_Transport_Mechanische_Stop/EM_Transport_Mechanische_Stop.TcPOU
FUNCTION_BLOCK EM_Transport_Mechanische_Stop EXTENDS EM_Transport IMPLEMENTS ITF_EM_Transport_Mechanische_Stop

VAR
	fbMechanischeStop_mem : STRUCT_EM_Mechanische_Stop;
	Klep		: CM_Valve;
END_VAR

(*
$$$$$$$$\                                                                   $$\       $$$$$$$$\                     $$\                                         $$\                     
$$  _____|                                                                  $$ |      $$  _____|                    \__|                                        \__|                    
$$ |   $$$$$$\   $$$$$$\  $$$$$$$\  $$\  $$\  $$\  $$$$$$\   $$$$$$\   $$$$$$$ |      $$ |      $$$$$$$\   $$$$$$\  $$\ $$$$$$$\   $$$$$$\   $$$$$$\   $$$$$$\  $$\ $$$$$$$\   $$$$$$\  
$$$$$\ \____$$\ $$  __$$\ $$  __$$\ $$ | $$ | $$ |$$  __$$\ $$  __$$\ $$  __$$ |      $$$$$\    $$  __$$\ $$  __$$\ $$ |$$  __$$\ $$  __$$\ $$  __$$\ $$  __$$\ $$ |$$  __$$\ $$  __$$\ 
$$  __|$$$$$$$ |$$ |  \__|$$ |  $$ |$$ | $$ | $$ |$$ /  $$ |$$ /  $$ |$$ /  $$ |      $$  __|   $$ |  $$ |$$ /  $$ |$$ |$$ |  $$ |$$$$$$$$ |$$$$$$$$ |$$ |  \__|$$ |$$ |  $$ |$$ /  $$ |
$$ |  $$  __$$ |$$ |      $$ |  $$ |$$ | $$ | $$ |$$ |  $$ |$$ |  $$ |$$ |  $$ |      $$ |      $$ |  $$ |$$ |  $$ |$$ |$$ |  $$ |$$   ____|$$   ____|$$ |      $$ |$$ |  $$ |$$ |  $$ |
$$ |  \$$$$$$$ |$$ |      $$ |  $$ |\$$$$$\$$$$  |\$$$$$$  |\$$$$$$  |\$$$$$$$ |      $$$$$$$$\ $$ |  $$ |\$$$$$$$ |$$ |$$ |  $$ |\$$$$$$$\ \$$$$$$$\ $$ |      $$ |$$ |  $$ |\$$$$$$$ |
\__|   \_______|\__|      \__|  \__| \_____\____/  \______/  \______/  \_______|      \________|\__|  \__| \____$$ |\__|\__|  \__| \_______| \_______|\__|      \__|\__|  \__| \____$$ |
                                                                                                          $$\   $$ |                                                          $$\   $$ |
                                                                                                          \$$$$$$  |                                                          \$$$$$$  |
                                                                                                           \______/                                                            \______/ 
*)

//********************************Init***********************************
Klep();
SUPER^();
										
//********************************ZEROING***********************************	
(*								
fb_mem.STS.Auto 			:= FALSE;
fb_mem.STS.Manueel 			:= FALSE;
fb_mem.STS.Starting_SC 		:= FALSE;
fb_mem.STS.Execute_SC 		:= FALSE;
fb_mem.STS.Resetting_SC 	:= FALSE;
fb_mem.STS.Holding_SC 		:= FALSE;
fb_mem.STS.Unholding_SC 	:= FALSE;
fb_mem.STS.Suspending_SC 	:= FALSE;
fb_mem.STS.Unsuspending_SC 	:= FALSE;
fb_mem.STS.Aborting_SC 		:= FALSE;
fb_mem.STS.Clearing_SC 		:= FALSE;
fb_mem.STS.Stopping_SC 		:= FALSE;
fb_mem.STS.Completing_SC 	:= FALSE;
*)

//********************************Auto manual logic***********************************


//********************************Exeptionhandling***********************************

//********************************Action case***********************************


//********************************ZEROING***********************************
//Control Signals 
(*
fb_mem.CS.Auto            := FALSE;
fb_mem.CS.Manueel         := FALSE;
fb_mem.CS.Start           := FALSE;
fb_mem.CS.Stop            := FALSE;
fb_mem.CS.Reset           := FALSE;
fb_mem.CS.Abort           := FALSE;
fb_mem.CS.Clear           := FALSE;
fb_mem.CS.UnSuspend       := FALSE;
fb_mem.CS.Suspend         := FALSE;
fb_mem.CS.UnHold          := FALSE;
fb_mem.CS.Hold            := FALSE;
*)

{warning 'add method implementation '}
METHOD Close : BOOL
END_METHOD

{warning 'add method implementation '}
METHOD Open : BOOL
END_METHOD

PROPERTY Stop_State : E_Mechanische_Stop
GET
Stop_State := fbMechanischeStop_mem.STS.State;
END_GET
END_PROPERTY

{warning 'add method implementation '}
METHOD ZeroAllValues : BOOL
END_METHOD

END_FUNCTION_BLOCK

// ---- POUs/2. Equipment Modules/4. EM_Transport/EM_Transport.TcPOU
FUNCTION_BLOCK EM_Transport IMPLEMENTS  ITF_EM_Transport, ITF_PackML

VAR
	fb_mem : STRUCT_EM_Transport;
	bFirstCycleExecuted	: BOOL;
	
	Motor		: CM_Motor;
	Sensor		: CM_Sensor;
	
	ton1		: ton;
END_VAR

(*
$$$$$$$$\                                                                   $$\       $$$$$$$$\                     $$\                                         $$\                     
$$  _____|                                                                  $$ |      $$  _____|                    \__|                                        \__|                    
$$ |   $$$$$$\   $$$$$$\  $$$$$$$\  $$\  $$\  $$\  $$$$$$\   $$$$$$\   $$$$$$$ |      $$ |      $$$$$$$\   $$$$$$\  $$\ $$$$$$$\   $$$$$$\   $$$$$$\   $$$$$$\  $$\ $$$$$$$\   $$$$$$\  
$$$$$\ \____$$\ $$  __$$\ $$  __$$\ $$ | $$ | $$ |$$  __$$\ $$  __$$\ $$  __$$ |      $$$$$\    $$  __$$\ $$  __$$\ $$ |$$  __$$\ $$  __$$\ $$  __$$\ $$  __$$\ $$ |$$  __$$\ $$  __$$\ 
$$  __|$$$$$$$ |$$ |  \__|$$ |  $$ |$$ | $$ | $$ |$$ /  $$ |$$ /  $$ |$$ /  $$ |      $$  __|   $$ |  $$ |$$ /  $$ |$$ |$$ |  $$ |$$$$$$$$ |$$$$$$$$ |$$ |  \__|$$ |$$ |  $$ |$$ /  $$ |
$$ |  $$  __$$ |$$ |      $$ |  $$ |$$ | $$ | $$ |$$ |  $$ |$$ |  $$ |$$ |  $$ |      $$ |      $$ |  $$ |$$ |  $$ |$$ |$$ |  $$ |$$   ____|$$   ____|$$ |      $$ |$$ |  $$ |$$ |  $$ |
$$ |  \$$$$$$$ |$$ |      $$ |  $$ |\$$$$$\$$$$  |\$$$$$$  |\$$$$$$  |\$$$$$$$ |      $$$$$$$$\ $$ |  $$ |\$$$$$$$ |$$ |$$ |  $$ |\$$$$$$$\ \$$$$$$$\ $$ |      $$ |$$ |  $$ |\$$$$$$$ |
\__|   \_______|\__|      \__|  \__| \_____\____/  \______/  \______/  \_______|      \________|\__|  \__| \____$$ |\__|\__|  \__| \_______| \_______|\__|      \__|\__|  \__| \____$$ |
                                                                                                          $$\   $$ |                                                          $$\   $$ |
                                                                                                          \$$$$$$  |                                                          \$$$$$$  |
                                                                                                           \______/                                                            \______/ 
*)//********************************Initiating***********************************
fb_mem.STS.State := PackML_StateMachine(State			:= fb_mem.STS.State,
										Start           := fb_mem.CS.Start,
										Stop            := fb_mem.CS.Stop,
										Reset           := fb_mem.CS.Reset,
										Abort           := fb_mem.CS.Abort,
										Clear           := fb_mem.CS.Clear,
										UnSuspend       := fb_mem.CS.UnSuspend,
										Suspend         := fb_mem.CS.Suspend,
										UnHold          := fb_mem.CS.UnHold,
										Hold            := fb_mem.CS.Hold,
										Starting_SC     := fb_mem.STS.Starting_SC,
										Execute_SC      := fb_mem.STS.Execute_SC,
										Completing_SC	:= fb_mem.STS.Completing_SC,
										Resetting_SC    := fb_mem.STS.Resetting_SC,
										Holding_SC      := fb_mem.STS.Holding_SC,
										Unholding_SC    := fb_mem.STS.Unholding_SC,
										Suspending_SC   := fb_mem.STS.Suspending_SC,
										Unsuspending_SC := fb_mem.STS.Unsuspending_SC,
										Aborting_SC     := fb_mem.STS.Aborting_SC,
										Clearing_SC     := fb_mem.STS.Clearing_SC,
										Stopping_SC     := fb_mem.STS.Stopping_SC);

//********************************Init***********************************
Motor();
Sensor();			
										
//********************************ZEROING***********************************
fb_mem.STS.Starting_SC 		:= FALSE;
fb_mem.STS.Execute_SC 		:= FALSE;
fb_mem.STS.Resetting_SC 	:= FALSE;
fb_mem.STS.Holding_SC 		:= FALSE;
fb_mem.STS.Unholding_SC 	:= FALSE;
fb_mem.STS.Suspending_SC 	:= FALSE;
fb_mem.STS.Unsuspending_SC 	:= FALSE;
fb_mem.STS.Aborting_SC 		:= FALSE;
fb_mem.STS.Clearing_SC 		:= FALSE;
fb_mem.STS.Stopping_SC 		:= FALSE;
fb_mem.STS.Completing_SC 	:= FALSE;

//********************************Auto manual logic***********************************
IF NOT bFirstCycleExecuted THEN
	Motor.Auto := TRUE;
	Sensor.Auto := TRUE;
	bFirstCycleExecuted := TRUE;
END_IF

IF fb_mem.CS.Auto OR fb_mem.HMI.Auto THEN
	fb_mem.STS.Auto := TRUE;
	fb_mem.STS.Manueel := FALSE;
END_IF

IF fb_mem.CS.Manueel OR fb_mem.HMI.Manueel THEN
	fb_mem.STS.Auto := FALSE;
	fb_mem.STS.Manueel := TRUE;
END_IF

//********************************Exeptionhandling***********************************

